NETWORK
TITLE = 218 - LCP81_C311_BG6314 - Compactor Lock In Pos. OS - Locked

       CALL #"LCP81_C311_BG6314"
       (
         CM_No := 218 ,
         Tab := 26 ,
         SubTab := 7 ,
         CfgType := 0 ,
         CfgInvert := True ,
         InputRaw := LCP81_C311_BG6314_DI_FbP ,
         SC_Local := SL_26_P ,
         CM_ALM := #ALM[209] ,
       );

NETWORK
TITLE = 219 - LCP81_C311_BG6315 - Compactor Lock Out Pos. OS - Unlocked

       CALL #"LCP81_C311_BG6315"
       (
         CM_No := 219 ,
         Tab := 26 ,
         SubTab := 7 ,
         CfgType := 0 ,
         CfgInvert := True ,
         InputRaw := LCP81_C311_BG6315_DI_FbN ,
         SC_Local := SL_26_P ,
         CM_ALM := #ALM[210] ,
       );

NETWORK
TITLE = 220 - LCP81_C311_BG6316 - Compactor Lock In Pos. DS - Locked

       CALL #"LCP81_C311_BG6316"
       (
         CM_No := 220 ,
         Tab := 26 ,
         SubTab := 7 ,
         CfgType := 0 ,
         CfgInvert := True ,
         InputRaw := LCP81_C311_BG6316_DI_FbP ,
         SC_Local := SL_26_P ,
         CM_ALM := #ALM[211] ,
       );

NETWORK
TITLE = 221 - LCP81_C311_BG6317 - Compactor Lock Out Pos. DS - Unlocked

       CALL #"LCP81_C311_BG6317"
       (
         CM_No := 221 ,
         Tab := 26 ,
         SubTab := 7 ,
         CfgType := 0 ,
         CfgInvert := True ,
         InputRaw := LCP81_C311_BG6317_DI_FbN ,
         SC_Local := SL_26_P ,
         CM_ALM := #ALM[212] ,
       );

NETWORK
TITLE = 222 - LCP81_ES01_SF6136 - Emergency Stop  - Dryer 1 Ratio Box CB.81-01

       CALL #"LCP81_ES01_SF6136"
       (
         CM_No := 222 ,
         Tab := 1 ,
         SubTab := 5 ,
         CfgType := 0 ,
         CfgInvert := True ,
         InputRaw := LCP81_ES01_SF6136_DI_ChA ,
         SC_Local := SL_01 ,
         CM_ALM := #ALM[213] ,
       );

NETWORK
TITLE = 223 - LCP81_ES01_SF6137 - Emergency Stop  - Former Fan area

       CALL #"LCP81_ES01_SF6137"
       (
         CM_No := 223 ,
         Tab := 1 ,
         SubTab := 5 ,
         CfgType := 0 ,
         CfgInvert := True ,
         InputRaw := LCP81_ES01_SF6137_DI_ChA ,
         SC_Local := SL_01 ,
         CM_ALM := #ALM[214] ,
       );

NETWORK
TITLE = 224 - LCP81_ES01_SF6138 - Emergency Stop  - Former Fan area

       CALL #"LCP81_ES01_SF6138"
       (
         CM_No := 224 ,
         Tab := 1 ,
         SubTab := 5 ,
         CfgType := 0 ,
         CfgInvert := True ,
         InputRaw := LCP81_ES01_SF6138_DI_ChA ,
         SC_Local := SL_01 ,
         CM_ALM := #ALM[215] ,
       );

NETWORK
TITLE = 225 - LCP81_ES01_SF6139 - Emergency Stop  - LCP81

       CALL #"LCP81_ES01_SF6139"
       (
         CM_No := 225 ,
         Tab := 1 ,
         SubTab := 5 ,
         CfgType := 0 ,
         CfgInvert := True ,
         InputRaw := LCP81_ES01_SF6139_DI_ChA ,
         SC_Local := SL_01 ,
         CM_ALM := #ALM[216] ,
       );

NETWORK
TITLE = 226 - LCP81_DC01_FC1000 - Power Feed Module 24VDC - Status

       CALL #"LCP81_DC01_FC1000"
       (
         CM_No := 226 ,
         Tab := 13 ,
         SubTab := 5 ,
         CfgType := 0 ,
         CfgInvert := True ,
         InputRaw := LCP81_DC01_FC1000_DI_Sts ,
         SC_Local := SL_13 ,
         CM_ALM := #ALM[217] ,
       );

NETWORK
TITLE = 227 - LCP81_IO_KF1000 - Point IO - EtherNet/IP Adapter

       CALL #"LCP81_IO_KF1000"
       (
         CM_No := 227 ,
         Tab := 13 ,
         SubTab := 5 ,
         CfgType := 0 ,
         CfgInvert := True ,
         InputRaw :=  ,
         SC_Local := SL_13 ,
         CM_ALM := #ALM[218] ,
       );

NETWORK
TITLE = 228 - LCP81_IO_KF2000 - Point IO 2nd - EtherNet/IP Adapter

       CALL #"LCP81_IO_KF2000"
       (
         CM_No := 228 ,
         Tab := 13 ,
         SubTab := 5 ,
         CfgType := 0 ,
         CfgInvert := True ,
         InputRaw :=  ,
         SC_Local := SL_13 ,
         CM_ALM := #ALM[219] ,
       );

NETWORK
TITLE = 229 - LCP81_IO_KF3047 - 24V DC 8-Point Safety Input Module - SDI

       CALL #"LCP81_IO_KF3047"
       (
         CM_No := 229 ,
         Tab := 13 ,
         SubTab := 5 ,
         CfgType := 0 ,
         CfgInvert := True ,
         InputRaw :=  ,
         SC_Local := SL_13 ,
         CM_ALM := #ALM[220] ,
       );

NETWORK
TITLE = 230 - LCP81_IO_KF3048 - 24V DC 8-Point Safety Input Module - SDI

       CALL #"LCP81_IO_KF3048"
       (
         CM_No := 230 ,
         Tab := 13 ,
         SubTab := 5 ,
         CfgType := 0 ,
         CfgInvert := True ,
         InputRaw :=  ,
         SC_Local := SL_13 ,
         CM_ALM := #ALM[221] ,
       );

NETWORK
TITLE = 231 - LCP91_A110_SF6141 - Filter 1 Zone 1 - Ex doors & Estop

       CALL #"LCP91_A110_SF6141"
       (
         CM_No := 231 ,
         Tab := 1 ,
         SubTab := 3 ,
         CfgType := 0 ,
         CfgInvert := True ,
         InputRaw := LCP91_A110_SF6141_DI_ChA ,
         SC_Local := SL_01 ,
         CM_ALM := #ALM[222] ,
       );

NETWORK
TITLE = 232 - LCP91_A110_BG7712 - Filter 1 Zone 2 - Top Door

       CALL #"LCP91_A110_BG7712"
       (
         CM_No := 232 ,
         Tab := 1 ,
         SubTab := 3 ,
         CfgType := 0 ,
         CfgInvert := True ,
         InputRaw := LCP91_A110_BG7712_DI_ChA ,
         SC_Local := SL_01 ,
         CM_ALM := #ALM[223] ,
       );

NETWORK
TITLE = 233 - LCP91_A110_BG7711 - Filter 1 Zone 3 - Bottom Doors

       CALL #"LCP91_A110_BG7711"
       (
         CM_No := 233 ,
         Tab := 1 ,
         SubTab := 3 ,
         CfgType := 0 ,
         CfgInvert := True ,
         InputRaw := LCP91_A110_BG7711_DI_ChA ,
         SC_Local := SL_01 ,
         CM_ALM := #ALM[224] ,
       );

NETWORK
TITLE = 234 - LCP91_ES01_SF6142 - Emergency Stop  - LCP91

       CALL #"LCP91_ES01_SF6142"
       (
         CM_No := 234 ,
         Tab := 1 ,
         SubTab := 3 ,
         CfgType := 0 ,
         CfgInvert := True ,
         InputRaw := LCP91_ES01_SF6142_DI_ChA ,
         SC_Local := SL_01 ,
         CM_ALM := #ALM[225] ,
       );

NETWORK
TITLE = 235 - LCP91_DC01_FC1000 - Power Feed Module 24VDC - Status

       CALL #"LCP91_DC01_FC1000"
       (
         CM_No := 235 ,
         Tab := 13 ,
         SubTab := 5 ,
         CfgType := 0 ,
         CfgInvert := True ,
         InputRaw := LCP91_DC01_FC1000_DI_Sts ,
         SC_Local := SL_13 ,
         CM_ALM := #ALM[226] ,
       );

NETWORK
TITLE = 236 - LCP91_IO_KF1000 - Point IO - EtherNet/IP Adapter

       CALL #"LCP91_IO_KF1000"
       (
         CM_No := 236 ,
         Tab := 13 ,
         SubTab := 5 ,
         CfgType := 0 ,
         CfgInvert := True ,
         InputRaw :=  ,
         SC_Local := SL_13 ,
         CM_ALM := #ALM[227] ,
       );

NETWORK
TITLE = 237 - LCP91_IO_KF3015 - 24V DC 8-Point Safety Input Module - SDI

       CALL #"LCP91_IO_KF3015"
       (
         CM_No := 237 ,
         Tab := 13 ,
         SubTab := 5 ,
         CfgType := 0 ,
         CfgInvert := True ,
         InputRaw :=  ,
         SC_Local := SL_13 ,
         CM_ALM := #ALM[228] ,
       );

NETWORK
TITLE = 238 - LCP91_IO_KF3016 - 24V DC 8-Point Safety Input Module - SDI

       CALL #"LCP91_IO_KF3016"
       (
         CM_No := 238 ,
         Tab := 13 ,
         SubTab := 5 ,
         CfgType := 0 ,
         CfgInvert := True ,
         InputRaw :=  ,
         SC_Local := SL_13 ,
         CM_ALM := #ALM[229] ,
       );

NETWORK
TITLE = 239 - LCP91_IO_KF3017 - 24V DC IO Link Master Module - IO Link

       CALL #"LCP91_IO_KF3017"
       (
         CM_No := 239 ,
         Tab := 13 ,
         SubTab := 5 ,
         CfgType := 0 ,
         CfgInvert := True ,
         InputRaw :=  ,
         SC_Local := SL_13 ,
         CM_ALM := #ALM[230] ,
       );

NETWORK
TITLE = 240 - LCP92_A210_CB.A210-14 - Control Box - Baghouse Filter 2

       CALL #"LCP92_A210_CB.A210-14"
       (
         CM_No := 240 ,
         Tab := 21 ,
         SubTab := 2 ,
         CfgType := 0 ,
         CfgInvert := True ,
         InputRaw :=  ,
         SC_Local := SL_01 ,
         CM_ALM := #ALM[231] ,
       );

NETWORK
TITLE = 241 - LCP92_A210_SF6144 - Filter 2 Zone 1 - Ex doors & Estop

       CALL #"LCP92_A210_SF6144"
       (
         CM_No := 241 ,
         Tab := 1 ,
         SubTab := 3 ,
         CfgType := 0 ,
         CfgInvert := True ,
         InputRaw := LCP92_A210_SF6144_DI_ChA ,
         SC_Local := SL_01 ,
         CM_ALM := #ALM[232] ,
       );

NETWORK
TITLE = 242 - LCP92_A210_CB.A210-15 - Control Box - Baghouse Filter 2

       CALL #"LCP92_A210_CB.A210-15"
       (
         CM_No := 242 ,
         Tab := 21 ,
         SubTab := 2 ,
         CfgType := 0 ,
         CfgInvert := True ,
         InputRaw :=  ,
         SC_Local := SL_01 ,
         CM_ALM := #ALM[233] ,
       );

NETWORK
TITLE = 243 - LCP92_A210_BG7732 - Filter 2 Zone 2 - Top Door

       CALL #"LCP92_A210_BG7732"
       (
         CM_No := 243 ,
         Tab := 1 ,
         SubTab := 3 ,
         CfgType := 0 ,
         CfgInvert := True ,
         InputRaw := LCP92_A210_BG7732_DI_ChA ,
         SC_Local := SL_01 ,
         CM_ALM := #ALM[234] ,
       );

NETWORK
TITLE = 244 - LCP92_A210_BG7731 - Filter 2 Zone 3 - Bottom Doors

       CALL #"LCP92_A210_BG7731"
       (
         CM_No := 244 ,
         Tab := 1 ,
         SubTab := 3 ,
         CfgType := 0 ,
         CfgInvert := True ,
         InputRaw := LCP92_A210_BG7731_DI_ChA ,
         SC_Local := SL_01 ,
         CM_ALM := #ALM[235] ,
       );

NETWORK
TITLE = 245 - LCP92_ES01_SF6145 - Emergency Stop  - LCP92

       CALL #"LCP92_ES01_SF6145"
       (
         CM_No := 245 ,
         Tab := 1 ,
         SubTab := 3 ,
         CfgType := 0 ,
         CfgInvert := True ,
         InputRaw := LCP92_ES01_SF6145_DI_ChA ,
         SC_Local := SL_01 ,
         CM_ALM := #ALM[236] ,
       );

NETWORK
TITLE = 246 - LCP92_DC01_FC1000 - Power Feed Module 24VDC - Status

       CALL #"LCP92_DC01_FC1000"
       (
         CM_No := 246 ,
         Tab := 13 ,
         SubTab := 5 ,
         CfgType := 0 ,
         CfgInvert := True ,
         InputRaw := LCP92_DC01_FC1000_DI_Flt ,
         SC_Local := SL_13 ,
         CM_ALM := #ALM[237] ,
       );

NETWORK
TITLE = 247 - LCP92_IO_KF1000 - Point IO - EtherNet/IP Adapter

       CALL #"LCP92_IO_KF1000"
       (
         CM_No := 247 ,
         Tab := 13 ,
         SubTab := 5 ,
         CfgType := 0 ,
         CfgInvert := True ,
         InputRaw :=  ,
         SC_Local := SL_13 ,
         CM_ALM := #ALM[238] ,
       );

NETWORK
TITLE = 248 - LCP92_IO_KF3013 - 24V DC 8-Point Safety Input Module - SDI

       CALL #"LCP92_IO_KF3013"
       (
         CM_No := 248 ,
         Tab := 13 ,
         SubTab := 5 ,
         CfgType := 0 ,
         CfgInvert := True ,
         InputRaw :=  ,
         SC_Local := SL_13 ,
         CM_ALM := #ALM[239] ,
       );

NETWORK
TITLE = 249 - LCP92_IO_KF3014 - 24V DC 8-Point Safety Input Module - SDI

       CALL #"LCP92_IO_KF3014"
       (
         CM_No := 249 ,
         Tab := 13 ,
         SubTab := 5 ,
         CfgType := 0 ,
         CfgInvert := True ,
         InputRaw :=  ,
         SC_Local := SL_13 ,
         CM_ALM := #ALM[240] ,
       );

NETWORK
TITLE = 250 - LCP92_IO_KF3015 - 24V DC IO Link Master Module - IO Link

       CALL #"LCP92_IO_KF3015"
       (
         CM_No := 250 ,
         Tab := 13 ,
         SubTab := 5 ,
         CfgType := 0 ,
         CfgInvert := True ,
         InputRaw :=  ,
         SC_Local := SL_13 ,
         CM_ALM := #ALM[241] ,
       );

NETWORK
TITLE = 251 - LCP93_A171_FN3771 - Humidifier 1 Fan 1  - Motor Disconnect

       CALL #"LCP93_A171_FN3771"
       (
         CM_No := 251 ,
         Tab := 22 ,
         SubTab := 4 ,
         CfgType := 0 ,
         CfgInvert := True ,
         InputRaw := LCP93_A171_FN3771_DI_Flt ,
         SC_Local := SL_22_P ,
         CM_ALM := #ALM[242] ,
       );

NETWORK
TITLE = 252 - LCP93_A172_FN3772 - Humidifier 1 Fan 2  - Motor Disconnect

       CALL #"LCP93_A172_FN3772"
       (
         CM_No := 252 ,
         Tab := 22 ,
         SubTab := 4 ,
         CfgType := 0 ,
         CfgInvert := True ,
         InputRaw := LCP93_A172_FN3772_DI_Flt ,
         SC_Local := SL_22_P ,
         CM_ALM := #ALM[243] ,
       );

NETWORK
TITLE = 253 - LCP93_A173_FN3773 - Humidifier 1 Fan 3  - Motor Disconnect

       CALL #"LCP93_A173_FN3773"
       (
         CM_No := 253 ,
         Tab := 22 ,
         SubTab := 4 ,
         CfgType := 0 ,
         CfgInvert := True ,
         InputRaw := LCP93_A173_FN3773_DI_Flt ,
         SC_Local := SL_22_P ,
         CM_ALM := #ALM[244] ,
       );

NETWORK
TITLE = 254 - LCP93_A174_FN3774 - Humidifier 1 Fan 4  - Motor Disconnect

       CALL #"LCP93_A174_FN3774"
       (
         CM_No := 254 ,
         Tab := 22 ,
         SubTab := 4 ,
         CfgType := 0 ,
         CfgInvert := True ,
         InputRaw := LCP93_A174_FN3774_DI_Flt ,
         SC_Local := SL_22_P ,
         CM_ALM := #ALM[245] ,
       );

NETWORK
TITLE = 255 - LCP93_A191_FN3781 - Humidifier 3 Fan 1  - Motor Disconnect

       CALL #"LCP93_A191_FN3781"
       (
         CM_No := 255 ,
         Tab := 22 ,
         SubTab := 5 ,
         CfgType := 0 ,
         CfgInvert := True ,
         InputRaw := LCP93_A191_FN3781_DI_Flt ,
         SC_Local := SL_22_P ,
         CM_ALM := #ALM[246] ,
       );

NETWORK
TITLE = 256 - LCP93_A192_FN3782 - Humidifier 3 Fan 2  - Motor Disconnect

       CALL #"LCP93_A192_FN3782"
       (
         CM_No := 256 ,
         Tab := 22 ,
         SubTab := 5 ,
         CfgType := 0 ,
         CfgInvert := True ,
         InputRaw := LCP93_A192_FN3782_DI_Flt ,
         SC_Local := SL_22_P ,
         CM_ALM := #ALM[247] ,
       );

NETWORK
TITLE = 257 - LCP93_A193_FN3783 - Humidifier 3 Fan 3 - Motor Disconnect

       CALL #"LCP93_A193_FN3783"
       (
         CM_No := 257 ,
         Tab := 22 ,
         SubTab := 5 ,
         CfgType := 0 ,
         CfgInvert := True ,
         InputRaw := LCP93_A193_FN3783_DI_Flt ,
         SC_Local := SL_22_P ,
         CM_ALM := #ALM[248] ,
       );

NETWORK
TITLE = 258 - LCP93_A194_FN3784 - Humidifier 3 Fan 4 - Motor Disconnect

       CALL #"LCP93_A194_FN3784"
       (
         CM_No := 258 ,
         Tab := 22 ,
         SubTab := 5 ,
         CfgType := 0 ,
         CfgInvert := True ,
         InputRaw := LCP93_A194_FN3784_DI_Flt ,
         SC_Local := SL_22_P ,
         CM_ALM := #ALM[249] ,
       );

NETWORK
TITLE = 259 - LCP93_A271_FN3786 - Humidifier 4 Fan 1  - Motor Disconnect

       CALL #"LCP93_A271_FN3786"
       (
         CM_No := 259 ,
         Tab := 22 ,
         SubTab := 5 ,
         CfgType := 0 ,
         CfgInvert := True ,
         InputRaw := LCP93_A271_FN3786_DI_Flt ,
         SC_Local := SL_22_P ,
         CM_ALM := #ALM[250] ,
       );

NETWORK
TITLE = 260 - LCP93_A272_FN3787 - Humidifier 4 Fan 2  - Motor Disconnect

       CALL #"LCP93_A272_FN3787"
       (
         CM_No := 260 ,
         Tab := 22 ,
         SubTab := 5 ,
         CfgType := 0 ,
         CfgInvert := True ,
         InputRaw := LCP93_A272_FN3787_DI_Flt ,
         SC_Local := SL_22_P ,
         CM_ALM := #ALM[251] ,
       );

NETWORK
TITLE = 261 - LCP93_A273_FN3788 - Humidifier 4 Fan 3  - Motor Disconnect

       CALL #"LCP93_A273_FN3788"
       (
         CM_No := 261 ,
         Tab := 22 ,
         SubTab := 5 ,
         CfgType := 0 ,
         CfgInvert := True ,
         InputRaw := LCP93_A273_FN3788_DI_Flt ,
         SC_Local := SL_22_P ,
         CM_ALM := #ALM[252] ,
       );

NETWORK
TITLE = 262 - LCP93_A274_FN3789 - Humidifier 4 Fan 4 - Motor Disconnect

       CALL #"LCP93_A274_FN3789"
       (
         CM_No := 262 ,
         Tab := 22 ,
         SubTab := 5 ,
         CfgType := 0 ,
         CfgInvert := True ,
         InputRaw := LCP93_A274_FN3789_DI_Flt ,
         SC_Local := SL_22_P ,
         CM_ALM := #ALM[253] ,
       );

NETWORK
TITLE = 263 - LCP93_A281_FN3791 - Humidifier 5 Fan 1  - Motor Disconnect

       CALL #"LCP93_A281_FN3791"
       (
         CM_No := 263 ,
         Tab := 22 ,
         SubTab := 6 ,
         CfgType := 0 ,
         CfgInvert := True ,
         InputRaw := LCP93_A281_FN3791_DI_Flt ,
         SC_Local := SL_22_P ,
         CM_ALM := #ALM[254] ,
       );

NETWORK
TITLE = 264 - LCP93_A282_FN3792 - Humidifier 5 Fan 2  - Motor Disconnect

       CALL #"LCP93_A282_FN3792"
       (
         CM_No := 264 ,
         Tab := 22 ,
         SubTab := 6 ,
         CfgType := 0 ,
         CfgInvert := True ,
         InputRaw := LCP93_A282_FN3792_DI_Flt ,
         SC_Local := SL_22_P ,
         CM_ALM := #ALM[255] ,
       );

NETWORK
TITLE = 265 - LCP93_A283_FN3793 - Humidifier 5 Fan 3  - Motor Disconnect

       CALL #"LCP93_A283_FN3793"
       (
         CM_No := 265 ,
         Tab := 22 ,
         SubTab := 6 ,
         CfgType := 0 ,
         CfgInvert := True ,
         InputRaw := LCP93_A283_FN3793_DI_Flt ,
         SC_Local := SL_22_P ,
         CM_ALM := #ALM[256] ,
       );

NETWORK
TITLE = 266 - LCP93_A284_FN3794 - Humidifier 5 Fan 4  - Motor Disconnect

       CALL #"LCP93_A284_FN3794"
       (
         CM_No := 266 ,
         Tab := 22 ,
         SubTab := 6 ,
         CfgType := 0 ,
         CfgInvert := True ,
         InputRaw := LCP93_A284_FN3794_DI_Flt ,
         SC_Local := SL_22_P ,
         CM_ALM := #ALM[257] ,
       );

NETWORK
TITLE = 267 - LCP93_A291_FN3796 - Humidifier 6 Fan 1  - Motor Disconnect

       CALL #"LCP93_A291_FN3796"
       (
         CM_No := 267 ,
         Tab := 22 ,
         SubTab := 6 ,
         CfgType := 0 ,
         CfgInvert := True ,
         InputRaw := LCP93_A291_FN3796_DI_Flt ,
         SC_Local := SL_22_P ,
         CM_ALM := #ALM[258] ,
       );

NETWORK
TITLE = 268 - LCP93_A292_FN3797 - Humidifier 6 Fan 2  - Motor Disconnect

       CALL #"LCP93_A292_FN3797"
       (
         CM_No := 268 ,
         Tab := 22 ,
         SubTab := 6 ,
         CfgType := 0 ,
         CfgInvert := True ,
         InputRaw := LCP93_A292_FN3797_DI_Flt ,
         SC_Local := SL_22_P ,
         CM_ALM := #ALM[259] ,
       );

NETWORK
TITLE = 269 - LCP93_A293_FN3798 - Humidifier 6 Fan 3  - Motor Disconnect

       CALL #"LCP93_A293_FN3798"
       (
         CM_No := 269 ,
         Tab := 22 ,
         SubTab := 6 ,
         CfgType := 0 ,
         CfgInvert := True ,
         InputRaw := LCP93_A293_FN3798_DI_Flt ,
         SC_Local := SL_22_P ,
         CM_ALM := #ALM[260] ,
       );

NETWORK
TITLE = 270 - LCP93_A294_FN3799 - Humidifier 6 Fan 4 - Motor Disconnect

       CALL #"LCP93_A294_FN3799"
       (
         CM_No := 270 ,
         Tab := 22 ,
         SubTab := 6 ,
         CfgType := 0 ,
         CfgInvert := True ,
         InputRaw := LCP93_A294_FN3799_DI_Flt ,
         SC_Local := SL_22_P ,
         CM_ALM := #ALM[261] ,
       );

NETWORK
TITLE = 271 - LCP93_A170_BG7830 - Door 1 Humidifier 1 - Fan Room

       CALL #"LCP93_A170_BG7830"
       (
         CM_No := 271 ,
         Tab := 1 ,
         SubTab := 3 ,
         CfgType := 0 ,
         CfgInvert := True ,
         InputRaw := LCP93_A170_BG7830_DI_ChA ,
         SC_Local := SL_22_P ,
         CM_ALM := #ALM[262] ,
       );

NETWORK
TITLE = 272 - LCP93_A190_BG7832 - Door 1 Humidifier 3 - Fan Room

       CALL #"LCP93_A190_BG7832"
       (
         CM_No := 272 ,
         Tab := 1 ,
         SubTab := 3 ,
         CfgType := 0 ,
         CfgInvert := True ,
         InputRaw := LCP93_A190_BG7832_DI_ChA ,
         SC_Local := SL_22_P ,
         CM_ALM := #ALM[263] ,
       );

NETWORK
TITLE = 273 - LCP93_A270_BG7834 - Door 1 Humidifier 4 - Fan Room

       CALL #"LCP93_A270_BG7834"
       (
         CM_No := 273 ,
         Tab := 1 ,
         SubTab := 3 ,
         CfgType := 0 ,
         CfgInvert := True ,
         InputRaw := LCP93_A270_BG7834_DI_ChA ,
         SC_Local := SL_22_P ,
         CM_ALM := #ALM[264] ,
       );

NETWORK
TITLE = 274 - LCP93_A280_BG7836 - Door 1 Humidifier 5 - Fan Room

       CALL #"LCP93_A280_BG7836"
       (
         CM_No := 274 ,
         Tab := 1 ,
         SubTab := 3 ,
         CfgType := 0 ,
         CfgInvert := True ,
         InputRaw := LCP93_A280_BG7836_DI_ChA ,
         SC_Local := SL_22_P ,
         CM_ALM := #ALM[265] ,
       );

NETWORK
TITLE = 275 - LCP93_A290_BG7838 - Door 1 Humidifier 6 - Fan Room

       CALL #"LCP93_A290_BG7838"
       (
         CM_No := 275 ,
         Tab := 1 ,
         SubTab := 3 ,
         CfgType := 0 ,
         CfgInvert := True ,
         InputRaw := LCP93_A290_BG7838_DI_ChA ,
         SC_Local := SL_22_P ,
         CM_ALM := #ALM[266] ,
       );

NETWORK
TITLE = 276 - LCP93_ES01_SF6146 - Emergency Stop  - Humidifier Area

       CALL #"LCP93_ES01_SF6146"
       (
         CM_No := 276 ,
         Tab := 1 ,
         SubTab := 3 ,
         CfgType := 0 ,
         CfgInvert := True ,
         InputRaw := LCP93_ES01_SF6146_DI_ChA ,
         SC_Local := SL_01 ,
         CM_ALM := #ALM[267] ,
       );

NETWORK
TITLE = 277 - LCP93_ES01_SF6147 - Emergency Stop  - Humidifier Area

       CALL #"LCP93_ES01_SF6147"
       (
         CM_No := 277 ,
         Tab := 1 ,
         SubTab := 3 ,
         CfgType := 0 ,
         CfgInvert := True ,
         InputRaw := LCP93_ES01_SF6147_DI_ChA ,
         SC_Local := SL_01 ,
         CM_ALM := #ALM[268] ,
       );

NETWORK
TITLE = 278 - LCP93_ES01_SF6148 - Emergency Stop  - Humidifier Area

       CALL #"LCP93_ES01_SF6148"
       (
         CM_No := 278 ,
         Tab := 1 ,
         SubTab := 3 ,
         CfgType := 0 ,
         CfgInvert := True ,
         InputRaw := LCP93_ES01_SF6148_DI_ChA ,
         SC_Local := SL_01 ,
         CM_ALM := #ALM[269] ,
       );

NETWORK
TITLE = 279 - LCP93_ES01_SF6149 - Emergency Stop  - LCP93

       CALL #"LCP93_ES01_SF6149"
       (
         CM_No := 279 ,
         Tab := 1 ,
         SubTab := 3 ,
         CfgType := 0 ,
         CfgInvert := True ,
         InputRaw := LCP93_ES01_SF6149_DI_ChA ,
         SC_Local := SL_01 ,
         CM_ALM := #ALM[270] ,
       );

NETWORK
TITLE = 280 - LCP93_DC01_FC1000 - Power Feed Module 24VDC - Status

       CALL #"LCP93_DC01_FC1000"
       (
         CM_No := 280 ,
         Tab := 13 ,
         SubTab := 5 ,
         CfgType := 0 ,
         CfgInvert := True ,
         InputRaw := LCP93_DC01_FC1000_DI_Flt ,
         SC_Local := SL_13 ,
         CM_ALM := #ALM[271] ,
       );

NETWORK
TITLE = 281 - LCP93_IO_KF1000 - Point IO - EtherNet/IP Adapter

       CALL #"LCP93_IO_KF1000"
       (
         CM_No := 281 ,
         Tab := 13 ,
         SubTab := 5 ,
         CfgType := 0 ,
         CfgInvert := True ,
         InputRaw :=  ,
         SC_Local := SL_13 ,
         CM_ALM := #ALM[272] ,
       );

NETWORK
TITLE = 282 - LCP93_IO_KF3020 - 24V DC 8-Point Safety Input Module - SDI

       CALL #"LCP93_IO_KF3020"
       (
         CM_No := 282 ,
         Tab := 13 ,
         SubTab := 5 ,
         CfgType := 0 ,
         CfgInvert := True ,
         InputRaw :=  ,
         SC_Local := SL_13 ,
         CM_ALM := #ALM[273] ,
       );

NETWORK
TITLE = 283 - LCP93_IO_KF3021 - 24V DC 8-Point Safety Input Module - SDI

       CALL #"LCP93_IO_KF3021"
       (
         CM_No := 283 ,
         Tab := 13 ,
         SubTab := 5 ,
         CfgType := 0 ,
         CfgInvert := True ,
         InputRaw :=  ,
         SC_Local := SL_13 ,
         CM_ALM := #ALM[274] ,
       );

NETWORK
TITLE = 284 - LCP93_IO_KF3022 - 24V DC 8-Point Safety Input Module - SDI

       CALL #"LCP93_IO_KF3022"
       (
         CM_No := 284 ,
         Tab := 13 ,
         SubTab := 5 ,
         CfgType := 0 ,
         CfgInvert := True ,
         InputRaw :=  ,
         SC_Local := SL_13 ,
         CM_ALM := #ALM[275] ,
       );

NETWORK
TITLE = 285 - LCP101_AC01_FC3101 - 115VAC Power Supply - Thermal Fault

       CALL #"LCP101_AC01_FC3101"
       (
         CM_No := 285 ,
         Tab := 13 ,
         SubTab := 6 ,
         CfgType := 0 ,
         CfgInvert := True ,
         InputRaw := LCP101_AC01_FC3101_DI_Flt ,
         SC_Local := SL_13 ,
         CM_ALM := #ALM[276] ,
       );

NETWORK
TITLE = 286 - LCP101_I610_QA1101 - Min Gas Pressure Switch - (-BP8101)

       CALL #"LCP101_I610_QA1101"
       (
         CM_No := 286 ,
         Tab := 28 ,
         SubTab := 3 ,
         CfgType := 0 ,
         CfgInvert := True ,
         InputRaw := LCP101_I610_QA1101_DI_FltL ,
         SC_Local := SL_28_S1 ,
         CM_ALM := #ALM[277] ,
       );

NETWORK
TITLE = 287 - LCP101_I610_QA1102 - Max Gas Pressure Switch - (-BP8102)

       CALL #"LCP101_I610_QA1102"
       (
         CM_No := 287 ,
         Tab := 28 ,
         SubTab := 3 ,
         CfgType := 0 ,
         CfgInvert := True ,
         InputRaw := LCP101_I610_QA1102_DI_FltH ,
         SC_Local := SL_28_S1 ,
         CM_ALM := #ALM[278] ,
       );

NETWORK
TITLE = 288 - LCP101_I610_QA1103 - Leak Gas Pressure Switch - (-BP8103)

       CALL #"LCP101_I610_QA1103"
       (
         CM_No := 288 ,
         Tab := 28 ,
         SubTab := 3 ,
         CfgType := 0 ,
         CfgInvert := True ,
         InputRaw := LCP101_I610_QA1103_DI_Ps ,
         SC_Local := SL_28_S1 ,
         CM_ALM := #ALM[279] ,
       );

NETWORK
TITLE = 289 - LCP101_I610_QA1113 - No Air Check Pressure Switch - (-BP2113)

       CALL #"LCP101_I610_QA1113"
       (
         CM_No := 289 ,
         Tab := 28 ,
         SubTab := 3 ,
         CfgType := 0 ,
         CfgInvert := True ,
         InputRaw := LCP101_I610_QA1113_DI_Ps ,
         SC_Local := SL_28_S1 ,
         CM_ALM := #ALM[280] ,
       );

NETWORK
TITLE = 290 - LCP101_I610_QA1108 - Burner Failure - Signal from Maxon

       CALL #"LCP101_I610_QA1108"
       (
         CM_No := 290 ,
         Tab := 28 ,
         SubTab := 3 ,
         CfgType := 0 ,
         CfgInvert := True ,
         InputRaw := LCP101_I610_QA1108_DI_Flt ,
         SC_Local := SL_28_S1 ,
         CM_ALM := #ALM[281] ,
       );

NETWORK
TITLE = 291 - LCP101_I610_QA1104 - High Temperature Failure - Signal from JUMO

       CALL #"LCP101_I610_QA1104"
       (
         CM_No := 291 ,
         Tab := 28 ,
         SubTab := 3 ,
         CfgType := 0 ,
         CfgInvert := True ,
         InputRaw := LCP101_I610_QA1104_DI_Flt ,
         SC_Local := SL_28_S1 ,
         CM_ALM := #ALM[282] ,
       );

NETWORK
TITLE = 292 - LCP101_I512_BG7101 - Disc Filter 1 Door 1 - Before Filter

       CALL #"LCP101_I512_BG7101"
       (
         CM_No := 292 ,
         Tab := 1 ,
         SubTab := 8 ,
         CfgType := 0 ,
         CfgInvert := True ,
         InputRaw := LCP101_I512_BG7101_DI_ChA ,
         SC_Local := SL_28_S1 ,
         CM_ALM := #ALM[283] ,
       );

NETWORK
TITLE = 293 - LCP101_I512_BG7103 - Disc Filter 1 Door 2 - After Filter

       CALL #"LCP101_I512_BG7103"
       (
         CM_No := 293 ,
         Tab := 1 ,
         SubTab := 8 ,
         CfgType := 0 ,
         CfgInvert := True ,
         InputRaw := LCP101_I512_BG7103_DI_ChA ,
         SC_Local := SL_28_S1 ,
         CM_ALM := #ALM[284] ,
       );

NETWORK
TITLE = 294 - LCP101_I611_BP1120 - Zone 1 Circulation Fan - Diff. Pressure Circ. Fan 1

       CALL #"LCP101_I611_BP1120"
       (
         CM_No := 294 ,
         Tab := 28 ,
         SubTab := 3 ,
         CfgType := 0 ,
         CfgInvert := True ,
         InputRaw := LCP101_I611_BP1120_DI_Ps ,
         SC_Local := SL_28_S1 ,
         CM_ALM := #ALM[285] ,
       );

NETWORK
TITLE = 295 - LCP101_ES01_SF6151 - Emergency Stop  - Dryer 1 Zone 1 Area

       CALL #"LCP101_ES01_SF6151"
       (
         CM_No := 295 ,
         Tab := 1 ,
         SubTab := 5 ,
         CfgType := 0 ,
         CfgInvert := True ,
         InputRaw := LCP101_ES01_SF6151_DI_ChA ,
         SC_Local := SL_01 ,
         CM_ALM := #ALM[286] ,
       );

NETWORK
TITLE = 296 - LCP101_ES01_SF6152 - Emergency Stop  - LCP101

       CALL #"LCP101_ES01_SF6152"
       (
         CM_No := 296 ,
         Tab := 1 ,
         SubTab := 5 ,
         CfgType := 0 ,
         CfgInvert := True ,
         InputRaw := LCP101_ES01_SF6152_DI_ChA ,
         SC_Local := SL_01 ,
         CM_ALM := #ALM[287] ,
       );

NETWORK
TITLE = 297 - LCP101_DC01_FC1000 - Power Feed Module 24VDC - Status

       CALL #"LCP101_DC01_FC1000"
       (
         CM_No := 297 ,
         Tab := 13 ,
         SubTab := 6 ,
         CfgType := 0 ,
         CfgInvert := True ,
         InputRaw := LCP101_DC01_FC1000_DI_Flt ,
         SC_Local := SL_13 ,
         CM_ALM := #ALM[288] ,
       );

NETWORK
TITLE = 298 - LCP101_IO_KF1000 - Point IO - EtherNet/IP Adapter

       CALL #"LCP101_IO_KF1000"
       (
         CM_No := 298 ,
         Tab := 13 ,
         SubTab := 6 ,
         CfgType := 0 ,
         CfgInvert := True ,
         InputRaw :=  ,
         SC_Local := SL_13 ,
         CM_ALM := #ALM[289] ,
       );

NETWORK
TITLE = 299 - LCP101_IO_KF3013 - 24V DC 8-Point Safety Input Module - SDI

       CALL #"LCP101_IO_KF3013"
       (
         CM_No := 299 ,
         Tab := 13 ,
         SubTab := 6 ,
         CfgType := 0 ,
         CfgInvert := True ,
         InputRaw :=  ,
         SC_Local := SL_13 ,
         CM_ALM := #ALM[290] ,
       );

NETWORK
TITLE = 300 - LCP101_IO_KF3014 - 24V DC 8-Point Safety Input Module - SDI

       CALL #"LCP101_IO_KF3014"
       (
         CM_No := 300 ,
         Tab := 13 ,
         SubTab := 6 ,
         CfgType := 0 ,
         CfgInvert := True ,
         InputRaw :=  ,
         SC_Local := SL_13 ,
         CM_ALM := #ALM[291] ,
       );

NETWORK
TITLE = 301 - LCP102_AC01_FC3201 - 115VAC Power Supply - Thermal Fault

       CALL #"LCP102_AC01_FC3201"
       (
         CM_No := 301 ,
         Tab := 13 ,
         SubTab := 6 ,
         CfgType := 0 ,
         CfgInvert := True ,
         InputRaw := LCP102_AC01_FC3201_DI_Flt ,
         SC_Local := SL_13 ,
         CM_ALM := #ALM[292] ,
       );

NETWORK
TITLE = 302 - LCP102_I522_BG7201 - Disc Filter 2 Door 1 - Before Filter

       CALL #"LCP102_I522_BG7201"
       (
         CM_No := 302 ,
         Tab := 1 ,
         SubTab := 8 ,
         CfgType := 0 ,
         CfgInvert := True ,
         InputRaw := LCP102_I522_BG7201_DI_ChA ,
         SC_Local := SL_28_S1 ,
         CM_ALM := #ALM[293] ,
       );

NETWORK
TITLE = 303 - LCP102_I522_BG7203 - Disc Filter 2 Door 1 - After Filter

       CALL #"LCP102_I522_BG7203"
       (
         CM_No := 303 ,
         Tab := 1 ,
         SubTab := 8 ,
         CfgType := 0 ,
         CfgInvert := True ,
         InputRaw := LCP102_I522_BG7203_DI_ChA ,
         SC_Local := SL_28_S1 ,
         CM_ALM := #ALM[294] ,
       );

NETWORK
TITLE = 304 - LCP102_I621_BP1222 - Zone 2 Circulation Fan - Diff. Pressure Circ. Fan 2

       CALL #"LCP102_I621_BP1222"
       (
         CM_No := 304 ,
         Tab := 28 ,
         SubTab := 4 ,
         CfgType := 0 ,
         CfgInvert := True ,
         InputRaw := LCP102_I621_BP1222_DI_Ps ,
         SC_Local := SL_28_S1 ,
         CM_ALM := #ALM[295] ,
       );

NETWORK
TITLE = 305 - LCP102_ES01_SF6253 - Emergency Stop  - Dryer 1 Zone 2 Area

       CALL #"LCP102_ES01_SF6253"
       (
         CM_No := 305 ,
         Tab := 1 ,
         SubTab := 5 ,
         CfgType := 0 ,
         CfgInvert := True ,
         InputRaw := LCP102_ES01_SF6253_DI_ChA ,
         SC_Local := SL_01 ,
         CM_ALM := #ALM[296] ,
       );

NETWORK
TITLE = 306 - LCP102_ES01_SF6254 - Emergency Stop  - LCP102

       CALL #"LCP102_ES01_SF6254"
       (
         CM_No := 306 ,
         Tab := 1 ,
         SubTab := 5 ,
         CfgType := 0 ,
         CfgInvert := True ,
         InputRaw := LCP102_ES01_SF6254_DI_ChA ,
         SC_Local := SL_01 ,
         CM_ALM := #ALM[297] ,
       );

NETWORK
TITLE = 307 - LCP102_DC01_FC1000 - Power Feed Module 24VDC - Status

       CALL #"LCP102_DC01_FC1000"
       (
         CM_No := 307 ,
         Tab := 13 ,
         SubTab := 6 ,
         CfgType := 0 ,
         CfgInvert := True ,
         InputRaw := LCP102_DC01_FC1000_DI_Flt ,
         SC_Local := SL_13 ,
         CM_ALM := #ALM[298] ,
       );

NETWORK
TITLE = 308 - LCP102_IO_KF1000 - Point IO - EtherNet/IP Adapter

       CALL #"LCP102_IO_KF1000"
       (
         CM_No := 308 ,
         Tab := 13 ,
         SubTab := 6 ,
         CfgType := 0 ,
         CfgInvert := True ,
         InputRaw :=  ,
         SC_Local := SL_13 ,
         CM_ALM := #ALM[299] ,
       );

NETWORK
TITLE = 309 - LCP102_IO_KF3008 - 24V DC 8-Point Safety Input Module - SDI

       CALL #"LCP102_IO_KF3008"
       (
         CM_No := 309 ,
         Tab := 13 ,
         SubTab := 6 ,
         CfgType := 0 ,
         CfgInvert := True ,
         InputRaw :=  ,
         SC_Local := SL_13 ,
         CM_ALM := #ALM[300] ,
       );

NETWORK
TITLE = 310 - LCP102_IO_KF3009 - 24V DC 8-Point Safety Input Module - SDI

       CALL #"LCP102_IO_KF3009"
       (
         CM_No := 310 ,
         Tab := 13 ,
         SubTab := 6 ,
         CfgType := 0 ,
         CfgInvert := True ,
         InputRaw :=  ,
         SC_Local := SL_13 ,
         CM_ALM := #ALM[301] ,
       );

NETWORK
TITLE = 311 - LCP102_IO_KF3010 - 24V DC 8-Point Source Safety Output Module - SDO

       CALL #"LCP102_IO_KF3010"
       (
         CM_No := 311 ,
         Tab := 13 ,
         SubTab := 6 ,
         CfgType := 0 ,
         CfgInvert := True ,
         InputRaw :=  ,
         SC_Local := SL_13 ,
         CM_ALM := #ALM[302] ,
       );

NETWORK
TITLE = 312 - LCP103_AC01_FC3301 - 115VAC Power Supply - Thermal Fault

       CALL #"LCP103_AC01_FC3301"
       (
         CM_No := 312 ,
         Tab := 13 ,
         SubTab := 6 ,
         CfgType := 0 ,
         CfgInvert := True ,
         InputRaw := LCP103_AC01_FC3301_DI_Flt ,
         SC_Local := SL_13 ,
         CM_ALM := #ALM[303] ,
       );

NETWORK
TITLE = 313 - LCP103_I630_QA1301 - Min Gas Pressure Switch - (-BP8301)

       CALL #"LCP103_I630_QA1301"
       (
         CM_No := 313 ,
         Tab := 28 ,
         SubTab := 5 ,
         CfgType := 0 ,
         CfgInvert := True ,
         InputRaw := LCP103_I630_QA1301_DI_FltL ,
         SC_Local := SL_28_S2 ,
         CM_ALM := #ALM[304] ,
       );

NETWORK
TITLE = 314 - LCP103_I630_QA1302 - Max Gas Pressure Switch - (-BP8302)

       CALL #"LCP103_I630_QA1302"
       (
         CM_No := 314 ,
         Tab := 28 ,
         SubTab := 5 ,
         CfgType := 0 ,
         CfgInvert := True ,
         InputRaw := LCP103_I630_QA1302_DI_FltH ,
         SC_Local := SL_28_S2 ,
         CM_ALM := #ALM[305] ,
       );

NETWORK
TITLE = 315 - LCP103_I630_QA1303 - Leak Gas Pressure Switch - (-BP8303)

       CALL #"LCP103_I630_QA1303"
       (
         CM_No := 315 ,
         Tab := 28 ,
         SubTab := 5 ,
         CfgType := 0 ,
         CfgInvert := True ,
         InputRaw := LCP103_I630_QA1303_DI_Ps ,
         SC_Local := SL_28_S2 ,
         CM_ALM := #ALM[306] ,
       );

NETWORK
TITLE = 316 - LCP103_I630_QA1313 - No Air Check Pressure Switch - (-BP2313)

       CALL #"LCP103_I630_QA1313"
       (
         CM_No := 316 ,
         Tab := 28 ,
         SubTab := 5 ,
         CfgType := 0 ,
         CfgInvert := True ,
         InputRaw := LCP103_I630_QA1313_DI_Ps ,
         SC_Local := SL_28_S2 ,
         CM_ALM := #ALM[307] ,
       );

NETWORK
TITLE = 317 - LCP103_I630_QA1308 - Burner Failure - Signal from Maxon

       CALL #"LCP103_I630_QA1308"
       (
         CM_No := 317 ,
         Tab := 28 ,
         SubTab := 5 ,
         CfgType := 0 ,
         CfgInvert := True ,
         InputRaw := LCP103_I630_QA1308_DI_Flt ,
         SC_Local := SL_28_S2 ,
         CM_ALM := #ALM[308] ,
       );

NETWORK
TITLE = 318 - LCP103_I630_QA1304 - High Temperature Failure - Signal from JUMO

       CALL #"LCP103_I630_QA1304"
       (
         CM_No := 318 ,
         Tab := 28 ,
         SubTab := 5 ,
         CfgType := 0 ,
         CfgInvert := True ,
         InputRaw := LCP103_I630_QA1304_DI_Flt ,
         SC_Local := SL_28_S2 ,
         CM_ALM := #ALM[309] ,
       );

NETWORK
TITLE = 319 - LCP103_K512_BG7301 - Disc Filter 3 Door 1 - Before Filter

       CALL #"LCP103_K512_BG7301"
       (
         CM_No := 319 ,
         Tab := 1 ,
         SubTab := 8 ,
         CfgType := 0 ,
         CfgInvert := True ,
         InputRaw := LCP103_K512_BG7301_DI_ChA ,
         SC_Local := SL_28_S2 ,
         CM_ALM := #ALM[310] ,
       );

NETWORK
TITLE = 320 - LCP103_K512_BG7303 - Disc Filter 3 Door 2 - After Filter

       CALL #"LCP103_K512_BG7303"
       (
         CM_No := 320 ,
         Tab := 1 ,
         SubTab := 8 ,
         CfgType := 0 ,
         CfgInvert := True ,
         InputRaw := LCP103_K512_BG7303_DI_ChA ,
         SC_Local := SL_28_S2 ,
         CM_ALM := #ALM[311] ,
       );

NETWORK
TITLE = 321 - LCP103_K611_BP1323 - Zone 3 Circulation Fan - Diff. Pressure Circ. Fan 3

       CALL #"LCP103_K611_BP1323"
       (
         CM_No := 321 ,
         Tab := 28 ,
         SubTab := 5 ,
         CfgType := 0 ,
         CfgInvert := True ,
         InputRaw := LCP103_K611_BP1323_DI_Ps ,
         SC_Local := SL_28_S2 ,
         CM_ALM := #ALM[312] ,
       );

NETWORK
TITLE = 322 - LCP103_ES01_SF6355 - Emergency Stop  - Dryer 2 Zone 3 Area

       CALL #"LCP103_ES01_SF6355"
       (
         CM_No := 322 ,
         Tab := 1 ,
         SubTab := 5 ,
         CfgType := 0 ,
         CfgInvert := True ,
         InputRaw := LCP103_ES01_SF6355_DI_ChA ,
         SC_Local := SL_01 ,
         CM_ALM := #ALM[313] ,
       );

NETWORK
TITLE = 323 - LCP103_ES01_SF6356 - Emergency Stop  - LCP103

       CALL #"LCP103_ES01_SF6356"
       (
         CM_No := 323 ,
         Tab := 1 ,
         SubTab := 5 ,
         CfgType := 0 ,
         CfgInvert := True ,
         InputRaw := LCP103_ES01_SF6356_DI_ChA ,
         SC_Local := SL_01 ,
         CM_ALM := #ALM[314] ,
       );

NETWORK
TITLE = 324 - LCP103_DC01_FC1000 - Power Feed Module 24VDC - Status

       CALL #"LCP103_DC01_FC1000"
       (
         CM_No := 324 ,
         Tab := 13 ,
         SubTab := 6 ,
         CfgType := 0 ,
         CfgInvert := True ,
         InputRaw := LCP103_DC01_FC1000_DI_Flt ,
         SC_Local := SL_13 ,
         CM_ALM := #ALM[315] ,
       );

NETWORK
TITLE = 325 - LCP103_IO_KF1000 - Point IO - EtherNet/IP Adapter

       CALL #"LCP103_IO_KF1000"
       (
         CM_No := 325 ,
         Tab := 13 ,
         SubTab := 6 ,
         CfgType := 0 ,
         CfgInvert := True ,
         InputRaw :=  ,
         SC_Local := SL_13 ,
         CM_ALM := #ALM[316] ,
       );

NETWORK
TITLE = 326 - LCP103_IO_KF3013 - 24V DC 8-Point Safety Input Module - SDI

       CALL #"LCP103_IO_KF3013"
       (
         CM_No := 326 ,
         Tab := 13 ,
         SubTab := 6 ,
         CfgType := 0 ,
         CfgInvert := True ,
         InputRaw :=  ,
         SC_Local := SL_13 ,
         CM_ALM := #ALM[317] ,
       );

NETWORK
TITLE = 327 - LCP103_IO_KF3014 - 24V DC 8-Point Safety Input Module - SDI

       CALL #"LCP103_IO_KF3014"
       (
         CM_No := 327 ,
         Tab := 13 ,
         SubTab := 6 ,
         CfgType := 0 ,
         CfgInvert := True ,
         InputRaw :=  ,
         SC_Local := SL_13 ,
         CM_ALM := #ALM[318] ,
       );

NETWORK
TITLE = 328 - LCP104_AC01_FC3401 - 115VAC Power Supply - Thermal Fault

       CALL #"LCP104_AC01_FC3401"
       (
         CM_No := 328 ,
         Tab := 13 ,
         SubTab := 6 ,
         CfgType := 0 ,
         CfgInvert := True ,
         InputRaw := LCP104_AC01_FC3401_DI_Flt ,
         SC_Local := SL_13 ,
         CM_ALM := #ALM[319] ,
       );

NETWORK
TITLE = 329 - LCP104_I640_QA1401 - Min Gas Pressure Switch - (-BP8401)

       CALL #"LCP104_I640_QA1401"
       (
         CM_No := 329 ,
         Tab := 28 ,
         SubTab := 6 ,
         CfgType := 0 ,
         CfgInvert := True ,
         InputRaw := LCP104_I640_QA1401_DI_FltL ,
         SC_Local := SL_28_S2 ,
         CM_ALM := #ALM[320] ,
       );

NETWORK
TITLE = 330 - LCP104_I640_QA1402 - Max Gas Pressure Switch - (-BP8402)

       CALL #"LCP104_I640_QA1402"
       (
         CM_No := 330 ,
         Tab := 28 ,
         SubTab := 6 ,
         CfgType := 0 ,
         CfgInvert := True ,
         InputRaw := LCP104_I640_QA1402_DI_FltH ,
         SC_Local := SL_28_S2 ,
         CM_ALM := #ALM[321] ,
       );

NETWORK
TITLE = 331 - LCP104_I640_QA1403 - Leak Gas Pressure Switch - (-BP8403)

       CALL #"LCP104_I640_QA1403"
       (
         CM_No := 331 ,
         Tab := 28 ,
         SubTab := 6 ,
         CfgType := 0 ,
         CfgInvert := True ,
         InputRaw := LCP104_I640_QA1403_DI_Ps ,
         SC_Local := SL_28_S2 ,
         CM_ALM := #ALM[322] ,
       );

NETWORK
TITLE = 332 - LCP104_I640_QA1413 - No Air Check Pressure Switch - (-BP2413)

       CALL #"LCP104_I640_QA1413"
       (
         CM_No := 332 ,
         Tab := 28 ,
         SubTab := 6 ,
         CfgType := 0 ,
         CfgInvert := True ,
         InputRaw := LCP104_I640_QA1413_DI_Ps ,
         SC_Local := SL_28_S2 ,
         CM_ALM := #ALM[323] ,
       );

NETWORK
TITLE = 333 - LCP104_I640_QA1408 - Burner Failure - Signal from Maxon

       CALL #"LCP104_I640_QA1408"
       (
         CM_No := 333 ,
         Tab := 28 ,
         SubTab := 6 ,
         CfgType := 0 ,
         CfgInvert := True ,
         InputRaw := LCP104_I640_QA1408_DI_Flt ,
         SC_Local := SL_28_S2 ,
         CM_ALM := #ALM[324] ,
       );

NETWORK
TITLE = 334 - LCP104_I640_QA1404 - High Temperature Failure - Signal from JUMO

       CALL #"LCP104_I640_QA1404"
       (
         CM_No := 334 ,
         Tab := 28 ,
         SubTab := 6 ,
         CfgType := 0 ,
         CfgInvert := True ,
         InputRaw := LCP104_I640_QA1404_DI_Flt ,
         SC_Local := SL_28_S2 ,
         CM_ALM := #ALM[325] ,
       );

NETWORK
TITLE = 335 - LCP104_K522_BG7401 - Disc Filter 4 Door 1 - Before Filter

       CALL #"LCP104_K522_BG7401"
       (
         CM_No := 335 ,
         Tab := 1 ,
         SubTab := 8 ,
         CfgType := 0 ,
         CfgInvert := True ,
         InputRaw := LCP104_K522_BG7401_DI_ChA ,
         SC_Local := SL_28_S2 ,
         CM_ALM := #ALM[326] ,
       );

NETWORK
TITLE = 336 - LCP104_K522_BG7403 - Disc Filter 4 Door 2 - After Filter

       CALL #"LCP104_K522_BG7403"
       (
         CM_No := 336 ,
         Tab := 1 ,
         SubTab := 8 ,
         CfgType := 0 ,
         CfgInvert := True ,
         InputRaw := LCP104_K522_BG7403_DI_ChA ,
         SC_Local := SL_28_S2 ,
         CM_ALM := #ALM[327] ,
       );

NETWORK
TITLE = 337 - LCP104_K621_BP1424 - Zone 4 Circulation Fan  - Diff. Pressure Circ. Fan 4

       CALL #"LCP104_K621_BP1424"
       (
         CM_No := 337 ,
         Tab := 28 ,
         SubTab := 6 ,
         CfgType := 0 ,
         CfgInvert := True ,
         InputRaw := LCP104_K621_BP1424_DI_Ps ,
         SC_Local := SL_28_S2 ,
         CM_ALM := #ALM[328] ,
       );

NETWORK
TITLE = 338 - LCP104_ES01_SF6457 - Emergency Stop  - Dryer 2 Zone 4 Area

       CALL #"LCP104_ES01_SF6457"
       (
         CM_No := 338 ,
         Tab := 1 ,
         SubTab := 5 ,
         CfgType := 0 ,
         CfgInvert := True ,
         InputRaw := LCP104_ES01_SF6457_DI_ChA ,
         SC_Local := SL_01 ,
         CM_ALM := #ALM[329] ,
       );

NETWORK
TITLE = 339 - LCP104_ES01_SF6458 - Emergency Stop  - LCP104

       CALL #"LCP104_ES01_SF6458"
       (
         CM_No := 339 ,
         Tab := 1 ,
         SubTab := 5 ,
         CfgType := 0 ,
         CfgInvert := True ,
         InputRaw := LCP104_ES01_SF6458_DI_ChA ,
         SC_Local := SL_01 ,
         CM_ALM := #ALM[330] ,
       );

NETWORK
TITLE = 340 - LCP104_DC01_FC1000 - Power Feed Module 24VDC - Status

       CALL #"LCP104_DC01_FC1000"
       (
         CM_No := 340 ,
         Tab := 13 ,
         SubTab := 6 ,
         CfgType := 0 ,
         CfgInvert := True ,
         InputRaw := LCP104_DC01_FC1000_DI_Flt ,
         SC_Local := SL_13 ,
         CM_ALM := #ALM[331] ,
       );

NETWORK
TITLE = 341 - LCP104_IO_KF1000 - Point IO - EtherNet/IP Adapter

       CALL #"LCP104_IO_KF1000"
       (
         CM_No := 341 ,
         Tab := 13 ,
         SubTab := 6 ,
         CfgType := 0 ,
         CfgInvert := True ,
         InputRaw :=  ,
         SC_Local := SL_13 ,
         CM_ALM := #ALM[332] ,
       );

NETWORK
TITLE = 342 - LCP104_IO_KF3013 - 24V DC 8-Point Safety Input Module - SDI

       CALL #"LCP104_IO_KF3013"
       (
         CM_No := 342 ,
         Tab := 13 ,
         SubTab := 6 ,
         CfgType := 0 ,
         CfgInvert := True ,
         InputRaw :=  ,
         SC_Local := SL_13 ,
         CM_ALM := #ALM[333] ,
       );

NETWORK
TITLE = 343 - LCP104_IO_KF3014 - 24V DC 8-Point Safety Input Module - SDI

       CALL #"LCP104_IO_KF3014"
       (
         CM_No := 343 ,
         Tab := 13 ,
         SubTab := 6 ,
         CfgType := 0 ,
         CfgInvert := True ,
         InputRaw :=  ,
         SC_Local := SL_13 ,
         CM_ALM := #ALM[334] ,
       );

NETWORK
TITLE = 344 - LCP111_AC01_FC3501 - 115VAC Power Supply - Thermal Fault

       CALL #"LCP111_AC01_FC3501"
       (
         CM_No := 344 ,
         Tab := 13 ,
         SubTab := 6 ,
         CfgType := 0 ,
         CfgInvert := True ,
         InputRaw := LCP111_AC01_FC3501_DI_Flt ,
         SC_Local := SL_13 ,
         CM_ALM := #ALM[335] ,
       );

NETWORK
TITLE = 345 - LCP111_I650_QA1501 - Min Gas Pressure Switch - (-BP8501)

       CALL #"LCP111_I650_QA1501"
       (
         CM_No := 345 ,
         Tab := 28 ,
         SubTab := 7 ,
         CfgType := 0 ,
         CfgInvert := True ,
         InputRaw := LCP111_I650_QA1501_DI_FltL ,
         SC_Local := SL_28_S3 ,
         CM_ALM := #ALM[336] ,
       );

NETWORK
TITLE = 346 - LCP111_I650_QA1502 - Max Gas Pressure Switch - (-BP8502)

       CALL #"LCP111_I650_QA1502"
       (
         CM_No := 346 ,
         Tab := 28 ,
         SubTab := 7 ,
         CfgType := 0 ,
         CfgInvert := True ,
         InputRaw := LCP111_I650_QA1502_DI_FltH ,
         SC_Local := SL_28_S3 ,
         CM_ALM := #ALM[337] ,
       );

NETWORK
TITLE = 347 - LCP111_I650_QA1503 - Leak Gas Pressure Switch - (-BP8503)

       CALL #"LCP111_I650_QA1503"
       (
         CM_No := 347 ,
         Tab := 28 ,
         SubTab := 7 ,
         CfgType := 0 ,
         CfgInvert := True ,
         InputRaw := LCP111_I650_QA1503_DI_Ps ,
         SC_Local := SL_28_S3 ,
         CM_ALM := #ALM[338] ,
       );

NETWORK
TITLE = 348 - LCP111_I650_QA1513 - No Air Check Pressure Switch - (-BP2513)

       CALL #"LCP111_I650_QA1513"
       (
         CM_No := 348 ,
         Tab := 28 ,
         SubTab := 7 ,
         CfgType := 0 ,
         CfgInvert := True ,
         InputRaw := LCP111_I650_QA1513_DI_Ps ,
         SC_Local := SL_28_S3 ,
         CM_ALM := #ALM[339] ,
       );

NETWORK
TITLE = 349 - LCP111_I650_QA1508 - Burner Failure - Signal from Maxon

       CALL #"LCP111_I650_QA1508"
       (
         CM_No := 349 ,
         Tab := 28 ,
         SubTab := 7 ,
         CfgType := 0 ,
         CfgInvert := True ,
         InputRaw := LCP111_I650_QA1508_DI_Flt ,
         SC_Local := SL_28_S3 ,
         CM_ALM := #ALM[340] ,
       );

NETWORK
TITLE = 350 - LCP111_I650_QA1504 - High Temperature Failure - Signal from JUMO

       CALL #"LCP111_I650_QA1504"
       (
         CM_No := 350 ,
         Tab := 28 ,
         SubTab := 7 ,
         CfgType := 0 ,
         CfgInvert := True ,
         InputRaw := LCP111_I650_QA1504_DI_Flt ,
         SC_Local := SL_28_S3 ,
         CM_ALM := #ALM[341] ,
       );

NETWORK
TITLE = 351 - LCP111_N512_BG7501 - Disc Filter 5 Door 1 - Before Filter

       CALL #"LCP111_N512_BG7501"
       (
         CM_No := 351 ,
         Tab := 1 ,
         SubTab := 8 ,
         CfgType := 0 ,
         CfgInvert := True ,
         InputRaw := LCP111_N512_BG7501_DI_ChA ,
         SC_Local := SL_28_S3 ,
         CM_ALM := #ALM[342] ,
       );

NETWORK
TITLE = 352 - LCP111_N512_BG7503 - Disc Filter 5 Door 2 - After Filter

       CALL #"LCP111_N512_BG7503"
       (
         CM_No := 352 ,
         Tab := 1 ,
         SubTab := 8 ,
         CfgType := 0 ,
         CfgInvert := True ,
         InputRaw := LCP111_N512_BG7503_DI_ChA ,
         SC_Local := SL_28_S3 ,
         CM_ALM := #ALM[343] ,
       );

NETWORK
TITLE = 353 - LCP111_N611_BP1525 - Zone 5 Circulation Fan  - Diff. Pressure Circ. Fan 5

       CALL #"LCP111_N611_BP1525"
       (
         CM_No := 353 ,
         Tab := 28 ,
         SubTab := 7 ,
         CfgType := 0 ,
         CfgInvert := True ,
         InputRaw := LCP111_N611_BP1525_DI_Ps ,
         SC_Local := SL_28_S3 ,
         CM_ALM := #ALM[344] ,
       );

NETWORK
TITLE = 354 - LCP111_ES01_SF6559 - Emergency Stop  - Dryer 3 Zone 5 Area

       CALL #"LCP111_ES01_SF6559"
       (
         CM_No := 354 ,
         Tab := 1 ,
         SubTab := 6 ,
         CfgType := 0 ,
         CfgInvert := True ,
         InputRaw := LCP111_ES01_SF6559_DI_ChA ,
         SC_Local := SL_01 ,
         CM_ALM := #ALM[345] ,
       );

NETWORK
TITLE = 355 - LCP111_ES01_SF6560 - Emergency Stop  - LCP111

       CALL #"LCP111_ES01_SF6560"
       (
         CM_No := 355 ,
         Tab := 1 ,
         SubTab := 6 ,
         CfgType := 0 ,
         CfgInvert := True ,
         InputRaw := LCP111_ES01_SF6560_DI_ChA ,
         SC_Local := SL_01 ,
         CM_ALM := #ALM[346] ,
       );

NETWORK
TITLE = 356 - LCP111_DC01_FC1000 - Power Feed Module 24VDC - Status

       CALL #"LCP111_DC01_FC1000"
       (
         CM_No := 356 ,
         Tab := 13 ,
         SubTab := 6 ,
         CfgType := 0 ,
         CfgInvert := True ,
         InputRaw := LCP111_DC01_FC1000_DI_Flt ,
         SC_Local := SL_13 ,
         CM_ALM := #ALM[347] ,
       );

NETWORK
TITLE = 357 - LCP111_IO_KF1000 - Point IO - EtherNet/IP Adapter

       CALL #"LCP111_IO_KF1000"
       (
         CM_No := 357 ,
         Tab := 13 ,
         SubTab := 6 ,
         CfgType := 0 ,
         CfgInvert := True ,
         InputRaw :=  ,
         SC_Local := SL_13 ,
         CM_ALM := #ALM[348] ,
       );

NETWORK
TITLE = 358 - LCP111_IO_KF3013 - 24V DC 8-Point Safety Input Module - SDI

       CALL #"LCP111_IO_KF3013"
       (
         CM_No := 358 ,
         Tab := 13 ,
         SubTab := 6 ,
         CfgType := 0 ,
         CfgInvert := True ,
         InputRaw :=  ,
         SC_Local := SL_13 ,
         CM_ALM := #ALM[349] ,
       );

NETWORK
TITLE = 359 - LCP111_IO_KF3014 - 24V DC 8-Point Safety Input Module - SDI

       CALL #"LCP111_IO_KF3014"
       (
         CM_No := 359 ,
         Tab := 13 ,
         SubTab := 6 ,
         CfgType := 0 ,
         CfgInvert := True ,
         InputRaw :=  ,
         SC_Local := SL_13 ,
         CM_ALM := #ALM[350] ,
       );

NETWORK
TITLE = 360 - LCP112_AC01_FC3601 - 115VAC Power Supply - Thermal Fault

       CALL #"LCP112_AC01_FC3601"
       (
         CM_No := 360 ,
         Tab := 13 ,
         SubTab := 6 ,
         CfgType := 0 ,
         CfgInvert := True ,
         InputRaw := LCP112_AC01_FC3601_DI_Flt ,
         SC_Local := SL_13 ,
         CM_ALM := #ALM[351] ,
       );

NETWORK
TITLE = 361 - LCP112_I660_QA1601 - Min Gas Pressure Switch - (-BP8601)

       CALL #"LCP112_I660_QA1601"
       (
         CM_No := 361 ,
         Tab := 28 ,
         SubTab := 8 ,
         CfgType := 0 ,
         CfgInvert := True ,
         InputRaw := LCP112_I660_QA1601_DI_FltL ,
         SC_Local := SL_28_S3 ,
         CM_ALM := #ALM[352] ,
       );

NETWORK
TITLE = 362 - LCP112_I660_QA1602 - Max Gas Pressure Switch - (-BP8602)

       CALL #"LCP112_I660_QA1602"
       (
         CM_No := 362 ,
         Tab := 28 ,
         SubTab := 8 ,
         CfgType := 0 ,
         CfgInvert := True ,
         InputRaw := LCP112_I660_QA1602_DI_FltH ,
         SC_Local := SL_28_S3 ,
         CM_ALM := #ALM[353] ,
       );

NETWORK
TITLE = 363 - LCP112_I660_QA1603 - Leak Gas Pressure Switch - (-BP8603)

       CALL #"LCP112_I660_QA1603"
       (
         CM_No := 363 ,
         Tab := 28 ,
         SubTab := 8 ,
         CfgType := 0 ,
         CfgInvert := True ,
         InputRaw := LCP112_I660_QA1603_DI_Ps ,
         SC_Local := SL_28_S3 ,
         CM_ALM := #ALM[354] ,
       );

NETWORK
TITLE = 364 - LCP112_I660_QA1613 - No Air Check Pressure Switch - (-BP2613)

       CALL #"LCP112_I660_QA1613"
       (
         CM_No := 364 ,
         Tab := 28 ,
         SubTab := 8 ,
         CfgType := 0 ,
         CfgInvert := True ,
         InputRaw := LCP112_I660_QA1613_DI_Ps ,
         SC_Local := SL_28_S3 ,
         CM_ALM := #ALM[355] ,
       );

NETWORK
TITLE = 365 - LCP112_I660_QA1608 - Burner Failure - Signal from Maxon

       CALL #"LCP112_I660_QA1608"
       (
         CM_No := 365 ,
         Tab := 28 ,
         SubTab := 8 ,
         CfgType := 0 ,
         CfgInvert := True ,
         InputRaw := LCP112_I660_QA1608_DI_Flt ,
         SC_Local := SL_28_S3 ,
         CM_ALM := #ALM[356] ,
       );

NETWORK
TITLE = 366 - LCP112_I660_QA1604 - High Temperature Failure - Signal from JUMO

       CALL #"LCP112_I660_QA1604"
       (
         CM_No := 366 ,
         Tab := 28 ,
         SubTab := 8 ,
         CfgType := 0 ,
         CfgInvert := True ,
         InputRaw := LCP112_I660_QA1604_DI_Flt ,
         SC_Local := SL_28_S3 ,
         CM_ALM := #ALM[357] ,
       );

NETWORK
TITLE = 367 - LCP112_N522_BG7601 - Disc Filter 6 Door 1 - Before Filter

       CALL #"LCP112_N522_BG7601"
       (
         CM_No := 367 ,
         Tab := 1 ,
         SubTab := 8 ,
         CfgType := 0 ,
         CfgInvert := True ,
         InputRaw := LCP112_N522_BG7601_DI_ChA ,
         SC_Local := SL_28_S3 ,
         CM_ALM := #ALM[358] ,
       );

NETWORK
TITLE = 368 - LCP112_N522_BG7603 - Disc Filter 6 Door 2 - After Filter

       CALL #"LCP112_N522_BG7603"
       (
         CM_No := 368 ,
         Tab := 1 ,
         SubTab := 8 ,
         CfgType := 0 ,
         CfgInvert := True ,
         InputRaw := LCP112_N522_BG7603_DI_ChA ,
         SC_Local := SL_28_S3 ,
         CM_ALM := #ALM[359] ,
       );

NETWORK
TITLE = 369 - LCP112_N621_BP1626 - Zone 6 Circulation Fan  - Diff. Pressure Circ. Fan 6

       CALL #"LCP112_N621_BP1626"
       (
         CM_No := 369 ,
         Tab := 28 ,
         SubTab := 8 ,
         CfgType := 0 ,
         CfgInvert := True ,
         InputRaw := LCP112_N621_BP1626_DI_Ps ,
         SC_Local := SL_28_S3 ,
         CM_ALM := #ALM[360] ,
       );

NETWORK
TITLE = 370 - LCP112_ES01_SF6661 - Emergency Stop  - Dryer 3 Zone 6Area

       CALL #"LCP112_ES01_SF6661"
       (
         CM_No := 370 ,
         Tab := 1 ,
         SubTab := 6 ,
         CfgType := 0 ,
         CfgInvert := True ,
         InputRaw := LCP112_ES01_SF6661_DI_ChA ,
         SC_Local := SL_01 ,
         CM_ALM := #ALM[361] ,
       );

NETWORK
TITLE = 371 - LCP112_ES01_SF6662 - Emergency Stop  - LCP112

       CALL #"LCP112_ES01_SF6662"
       (
         CM_No := 371 ,
         Tab := 1 ,
         SubTab := 6 ,
         CfgType := 0 ,
         CfgInvert := True ,
         InputRaw := LCP112_ES01_SF6662_DI_ChA ,
         SC_Local := SL_01 ,
         CM_ALM := #ALM[362] ,
       );

NETWORK
TITLE = 372 - LCP112_DC01_FC1000 - Power Feed Module 24VDC - Status

       CALL #"LCP112_DC01_FC1000"
       (
         CM_No := 372 ,
         Tab := 13 ,
         SubTab := 6 ,
         CfgType := 0 ,
         CfgInvert := True ,
         InputRaw := LCP112_DC01_FC1000_DI_Flt ,
         SC_Local := SL_13 ,
         CM_ALM := #ALM[363] ,
       );

NETWORK
TITLE = 373 - LCP112_IO_KF1000 - Point IO - EtherNet/IP Adapter

       CALL #"LCP112_IO_KF1000"
       (
         CM_No := 373 ,
         Tab := 13 ,
         SubTab := 6 ,
         CfgType := 0 ,
         CfgInvert := True ,
         InputRaw :=  ,
         SC_Local := SL_13 ,
         CM_ALM := #ALM[364] ,
       );

NETWORK
TITLE = 374 - LCP112_IO_KF3013 - 24V DC 8-Point Safety Input Module - SDI

       CALL #"LCP112_IO_KF3013"
       (
         CM_No := 374 ,
         Tab := 13 ,
         SubTab := 6 ,
         CfgType := 0 ,
         CfgInvert := True ,
         InputRaw :=  ,
         SC_Local := SL_13 ,
         CM_ALM := #ALM[365] ,
       );

NETWORK
TITLE = 375 - LCP112_IO_KF3014 - 24V DC 8-Point Safety Input Module - SDI

       CALL #"LCP112_IO_KF3014"
       (
         CM_No := 375 ,
         Tab := 13 ,
         SubTab := 6 ,
         CfgType := 0 ,
         CfgInvert := True ,
         InputRaw :=  ,
         SC_Local := SL_13 ,
         CM_ALM := #ALM[366] ,
       );

NETWORK
TITLE = 376 - LCP113_AC01_FC3701 - 115VAC Power Supply - Thermal Fault

       CALL #"LCP113_AC01_FC3701"
       (
         CM_No := 376 ,
         Tab := 13 ,
         SubTab := 6 ,
         CfgType := 0 ,
         CfgInvert := True ,
         InputRaw := LCP113_AC01_FC3701_DI_Flt ,
         SC_Local := SL_13 ,
         CM_ALM := #ALM[367] ,
       );

NETWORK
TITLE = 377 - LCP113_I670_QA1701 - Min Gas Pressure Switch - (-BP8701)

       CALL #"LCP113_I670_QA1701"
       (
         CM_No := 377 ,
         Tab := 28 ,
         SubTab := 9 ,
         CfgType := 0 ,
         CfgInvert := True ,
         InputRaw := LCP113_I670_QA1701_DI_FltL ,
         SC_Local := SL_28_S3 ,
         CM_ALM := #ALM[368] ,
       );

NETWORK
TITLE = 378 - LCP113_I670_QA1702 - Max Gas Pressure Switch - (-BP8702)

       CALL #"LCP113_I670_QA1702"
       (
         CM_No := 378 ,
         Tab := 28 ,
         SubTab := 9 ,
         CfgType := 0 ,
         CfgInvert := True ,
         InputRaw := LCP113_I670_QA1702_DI_FltH ,
         SC_Local := SL_28_S3 ,
         CM_ALM := #ALM[369] ,
       );

NETWORK
TITLE = 379 - LCP113_I670_QA1703 - Leak Gas Pressure Switch - (-BP8703)

       CALL #"LCP113_I670_QA1703"
       (
         CM_No := 379 ,
         Tab := 28 ,
         SubTab := 9 ,
         CfgType := 0 ,
         CfgInvert := True ,
         InputRaw := LCP113_I670_QA1703_DI_Ps ,
         SC_Local := SL_28_S3 ,
         CM_ALM := #ALM[370] ,
       );

NETWORK
TITLE = 380 - LCP113_I670_QA1713 - No Air Check Pressure Switch - (-BP2713)

       CALL #"LCP113_I670_QA1713"
       (
         CM_No := 380 ,
         Tab := 28 ,
         SubTab := 9 ,
         CfgType := 0 ,
         CfgInvert := True ,
         InputRaw := LCP113_I670_QA1713_DI_Ps ,
         SC_Local := SL_28_S3 ,
         CM_ALM := #ALM[371] ,
       );

NETWORK
TITLE = 381 - LCP113_I670_QA1708 - Burner Failure - Signal from Maxon

       CALL #"LCP113_I670_QA1708"
       (
         CM_No := 381 ,
         Tab := 28 ,
         SubTab := 9 ,
         CfgType := 0 ,
         CfgInvert := True ,
         InputRaw := LCP113_I670_QA1708_DI_Flt ,
         SC_Local := SL_28_S3 ,
         CM_ALM := #ALM[372] ,
       );

NETWORK
TITLE = 382 - LCP113_I670_QA1704 - High Temperature Failure - Signal from JUMO

       CALL #"LCP113_I670_QA1704"
       (
         CM_No := 382 ,
         Tab := 28 ,
         SubTab := 9 ,
         CfgType := 0 ,
         CfgInvert := True ,
         InputRaw := LCP113_I670_QA1704_DI_Flt ,
         SC_Local := SL_28_S3 ,
         CM_ALM := #ALM[373] ,
       );

NETWORK
TITLE = 383 - LCP113_N532_BG7701 - Disc Filter 7 Door 1 - Before Filter

       CALL #"LCP113_N532_BG7701"
       (
         CM_No := 383 ,
         Tab := 1 ,
         SubTab := 8 ,
         CfgType := 0 ,
         CfgInvert := True ,
         InputRaw := LCP113_N532_BG7701_DI_ChA ,
         SC_Local := SL_28_S3 ,
         CM_ALM := #ALM[374] ,
       );

NETWORK
TITLE = 384 - LCP113_N532_BG7703 - Disc Filter 7 Door 2 - After Filter

       CALL #"LCP113_N532_BG7703"
       (
         CM_No := 384 ,
         Tab := 1 ,
         SubTab := 8 ,
         CfgType := 0 ,
         CfgInvert := True ,
         InputRaw := LCP113_N532_BG7703_DI_ChA ,
         SC_Local := SL_28_S3 ,
         CM_ALM := #ALM[375] ,
       );

NETWORK
TITLE = 385 - LCP113_N631_BP1727 - Zone 7 Circulation Fan - Diff. Pressure Circ. Fan 7

       CALL #"LCP113_N631_BP1727"
       (
         CM_No := 385 ,
         Tab := 28 ,
         SubTab := 9 ,
         CfgType := 0 ,
         CfgInvert := True ,
         InputRaw := LCP113_N631_BP1727_DI_Ps ,
         SC_Local := SL_28_S3 ,
         CM_ALM := #ALM[376] ,
       );

NETWORK
TITLE = 386 - LCP113_ES01_SF6762 - Emergency Stop  - Dryer 3 Zone 7 Area

       CALL #"LCP113_ES01_SF6762"
       (
         CM_No := 386 ,
         Tab := 1 ,
         SubTab := 6 ,
         CfgType := 0 ,
         CfgInvert := True ,
         InputRaw := LCP113_ES01_SF6762_DI_ChA ,
         SC_Local := SL_01 ,
         CM_ALM := #ALM[377] ,
       );

NETWORK
TITLE = 387 - LCP113_ES01_SF6763 - Emergency Stop  - LCP113

       CALL #"LCP113_ES01_SF6763"
       (
         CM_No := 387 ,
         Tab := 1 ,
         SubTab := 6 ,
         CfgType := 0 ,
         CfgInvert := True ,
         InputRaw := LCP113_ES01_SF6763_DI_ChA ,
         SC_Local := SL_01 ,
         CM_ALM := #ALM[378] ,
       );

NETWORK
TITLE = 388 - LCP113_DC01_FC1000 - Power Feed Module 24VDC - Status

       CALL #"LCP113_DC01_FC1000"
       (
         CM_No := 388 ,
         Tab := 13 ,
         SubTab := 6 ,
         CfgType := 0 ,
         CfgInvert := True ,
         InputRaw := LCP113_DC01_FC1000_DI_Flt ,
         SC_Local := SL_13 ,
         CM_ALM := #ALM[379] ,
       );

NETWORK
TITLE = 389 - LCP113_IO_KF1000 - Point IO - EtherNet/IP Adapter

       CALL #"LCP113_IO_KF1000"
       (
         CM_No := 389 ,
         Tab := 13 ,
         SubTab := 6 ,
         CfgType := 0 ,
         CfgInvert := True ,
         InputRaw :=  ,
         SC_Local := SL_13 ,
         CM_ALM := #ALM[380] ,
       );

NETWORK
TITLE = 390 - LCP113_IO_KF3013 - 24V DC 8-Point Safety Input Module - SDI

       CALL #"LCP113_IO_KF3013"
       (
         CM_No := 390 ,
         Tab := 13 ,
         SubTab := 6 ,
         CfgType := 0 ,
         CfgInvert := True ,
         InputRaw :=  ,
         SC_Local := SL_13 ,
         CM_ALM := #ALM[381] ,
       );

NETWORK
TITLE = 391 - LCP113_IO_KF3014 - 24V DC 8-Point Safety Input Module - SDI

       CALL #"LCP113_IO_KF3014"
       (
         CM_No := 391 ,
         Tab := 13 ,
         SubTab := 6 ,
         CfgType := 0 ,
         CfgInvert := True ,
         InputRaw :=  ,
         SC_Local := SL_13 ,
         CM_ALM := #ALM[382] ,
       );

NETWORK
TITLE = 392 - LCP121_ES01_SF6181 - Emergency Stop  - CB.121-01

       CALL #"LCP121_ES01_SF6181"
       (
         CM_No := 392 ,
         Tab := 1 ,
         SubTab := 7 ,
         CfgType := 0 ,
         CfgInvert := True ,
         InputRaw := LCP121_ES01_SF6181_DI_ChA ,
         SC_Local := SL_01 ,
         CM_ALM := #ALM[383] ,
       );

NETWORK
TITLE = 393 - LCP121_ES01_SF6182 - Emergency Stop  - CB.121-02

       CALL #"LCP121_ES01_SF6182"
       (
         CM_No := 393 ,
         Tab := 1 ,
         SubTab := 7 ,
         CfgType := 0 ,
         CfgInvert := True ,
         InputRaw := LCP121_ES01_SF6182_DI_ChA ,
         SC_Local := SL_01 ,
         CM_ALM := #ALM[384] ,
       );

NETWORK
TITLE = 394 - LCP121_DC01_FC1000 - Power Feed Module 24VDC - Status

       CALL #"LCP121_DC01_FC1000"
       (
         CM_No := 394 ,
         Tab := 13 ,
         SubTab := 7 ,
         CfgType := 0 ,
         CfgInvert := True ,
         InputRaw := LCP121_DC01_FC1000_DI_Flt ,
         SC_Local := SL_13 ,
         CM_ALM := #ALM[385] ,
       );

NETWORK
TITLE = 395 - LCP122_ES01_SF6184 - Emergency Stop  - CB122-01

       CALL #"LCP122_ES01_SF6184"
       (
         CM_No := 395 ,
         Tab := 1 ,
         SubTab := 7 ,
         CfgType := 0 ,
         CfgInvert := True ,
         InputRaw := LCP122_ES01_SF6184_DI_ChA ,
         SC_Local := SL_01 ,
         CM_ALM := #ALM[386] ,
       );

NETWORK
TITLE = 396 - LCP122_ES01_SF6185 - Emergency Stop  - CB122-02

       CALL #"LCP122_ES01_SF6185"
       (
         CM_No := 396 ,
         Tab := 1 ,
         SubTab := 7 ,
         CfgType := 0 ,
         CfgInvert := True ,
         InputRaw := LCP122_ES01_SF6185_DI_ChA ,
         SC_Local := SL_01 ,
         CM_ALM := #ALM[387] ,
       );

NETWORK
TITLE = 397 - LCP122_ES01_SF6186 - Emergency Stop  - CB.122-03

       CALL #"LCP122_ES01_SF6186"
       (
         CM_No := 397 ,
         Tab := 1 ,
         SubTab := 7 ,
         CfgType := 0 ,
         CfgInvert := True ,
         InputRaw := LCP122_ES01_SF6186_DI_ChA ,
         SC_Local := SL_01 ,
         CM_ALM := #ALM[388] ,
       );

NETWORK
TITLE = 398 - LCP122_DC01_FC1000 - Power Feed Module 24VDC - Status

       CALL #"LCP122_DC01_FC1000"
       (
         CM_No := 398 ,
         Tab := 13 ,
         SubTab := 7 ,
         CfgType := 0 ,
         CfgInvert := True ,
         InputRaw := LCP122_DC01_FC1000_DI_Flt ,
         SC_Local := SL_13 ,
         CM_ALM := #ALM[389] ,
       );

NETWORK
TITLE = 399 - LCP123_ES01_SF6188 - Emergency Stop  - CB.123-01

       CALL #"LCP123_ES01_SF6188"
       (
         CM_No := 399 ,
         Tab := 1 ,
         SubTab := 7 ,
         CfgType := 0 ,
         CfgInvert := True ,
         InputRaw := LCP123_ES01_SF6188_DI_ChA ,
         SC_Local := SL_01 ,
         CM_ALM := #ALM[390] ,
       );

NETWORK
TITLE = 400 - LCP122_ES01_SF6190 - Emergency Stop  - CB.122-04

       CALL #"LCP122_ES01_SF6190"
       (
         CM_No := 400 ,
         Tab := 1 ,
         SubTab := 7 ,
         CfgType := 0 ,
         CfgInvert := True ,
         InputRaw := LCP122_ES01_SF6190_DI_ChA ,
         SC_Local := SL_01 ,
         CM_ALM := #ALM[391] ,
       );

NETWORK
TITLE = 401 - LCP123_DC01_FC1000 - Power Feed Module 24VDC - Status

       CALL #"LCP123_DC01_FC1000"
       (
         CM_No := 401 ,
         Tab := 13 ,
         SubTab := 7 ,
         CfgType := 0 ,
         CfgInvert := True ,
         InputRaw := LCP123_DC01_FC1000_DI_Flt ,
         SC_Local := SL_13 ,
         CM_ALM := #ALM[392] ,
       );

NETWORK
TITLE = 402 - LCP121_IO_KF1000 - Point IO - EtherNet/IP Adapter

       CALL #"LCP121_IO_KF1000"
       (
         CM_No := 402 ,
         Tab := 13 ,
         SubTab := 5 ,
         CfgType := 0 ,
         CfgInvert := True ,
         InputRaw :=  ,
         SC_Local := SL_13 ,
         CM_ALM := #ALM[393] ,
       );

NETWORK
TITLE = 403 - LCP121_IO_KF3010 - 24V DC 8-Point Safety Input Module - SDI

       CALL #"LCP121_IO_KF3010"
       (
         CM_No := 403 ,
         Tab := 13 ,
         SubTab := 5 ,
         CfgType := 0 ,
         CfgInvert := True ,
         InputRaw :=  ,
         SC_Local := SL_13 ,
         CM_ALM := #ALM[394] ,
       );

NETWORK
TITLE = 404 - LCP131_I811_BP1201 - Zone 1 Burner Fan - Differential Pressure Sensor

       CALL #"LCP131_I811_BP1201"
       (
         CM_No := 404 ,
         Tab := 28 ,
         SubTab := 3 ,
         CfgType := 0 ,
         CfgInvert := True ,
         InputRaw := LCP131_I811_BP1201_DI_Ps ,
         SC_Local := SL_28_S1 ,
         CM_ALM := #ALM[395] ,
       );

NETWORK
TITLE = 405 - LCP131_K811_BP1202 - Zone 3 Burner Fan - Differential Pressure Sensor

       CALL #"LCP131_K811_BP1202"
       (
         CM_No := 405 ,
         Tab := 28 ,
         SubTab := 5 ,
         CfgType := 0 ,
         CfgInvert := True ,
         InputRaw := LCP131_K811_BP1202_DI_Ps ,
         SC_Local := SL_28_S2 ,
         CM_ALM := #ALM[396] ,
       );

NETWORK
TITLE = 406 - LCP131_K821_BP1203 - Zone 4 Burner Fan - Differential Pressure Sensor

       CALL #"LCP131_K821_BP1203"
       (
         CM_No := 406 ,
         Tab := 28 ,
         SubTab := 6 ,
         CfgType := 0 ,
         CfgInvert := True ,
         InputRaw := LCP131_K821_BP1203_DI_Ps ,
         SC_Local := SL_28_S2 ,
         CM_ALM := #ALM[397] ,
       );

NETWORK
TITLE = 407 - LCP131_N811_BP1204 - Zone 5 Burner Fan - Differential Pressure Sensor

       CALL #"LCP131_N811_BP1204"
       (
         CM_No := 407 ,
         Tab := 28 ,
         SubTab := 7 ,
         CfgType := 0 ,
         CfgInvert := True ,
         InputRaw := LCP131_N811_BP1204_DI_Ps ,
         SC_Local := SL_28_S3 ,
         CM_ALM := #ALM[398] ,
       );

NETWORK
TITLE = 408 - LCP131_N821_BP1205 - Zone 6 Burner Fan - Differential Pressure Sensor

       CALL #"LCP131_N821_BP1205"
       (
         CM_No := 408 ,
         Tab := 28 ,
         SubTab := 8 ,
         CfgType := 0 ,
         CfgInvert := True ,
         InputRaw := LCP131_N821_BP1205_DI_Ps ,
         SC_Local := SL_28_S3 ,
         CM_ALM := #ALM[399] ,
       );

NETWORK
TITLE = 409 - LCP131_N831_BP1206 - Zone 7 Burner Fan - Differential Pressure Sensor

       CALL #"LCP131_N831_BP1206"
       (
         CM_No := 409 ,
         Tab := 28 ,
         SubTab := 9 ,
         CfgType := 0 ,
         CfgInvert := True ,
         InputRaw := LCP131_N831_BP1206_DI_Ps ,
         SC_Local := SL_28_S3 ,
         CM_ALM := #ALM[400] ,
       );

NETWORK
TITLE = 410 - LCP131_I711_BP1207 - Exhaust Fan 1 - Differential Pressure Sensor

       CALL #"LCP131_I711_BP1207"
       (
         CM_No := 410 ,
         Tab := 28 ,
         SubTab := 3 ,
         CfgType := 0 ,
         CfgInvert := True ,
         InputRaw := LCP131_I711_BP1207_DI_Ps ,
         SC_Local := SL_28_S1 ,
         CM_ALM := #ALM[401] ,
       );

NETWORK
TITLE = 411 - LCP131_K711_BP1208 - Exhaust Fan 3 - Differential Pressure Sensor

       CALL #"LCP131_K711_BP1208"
       (
         CM_No := 411 ,
         Tab := 28 ,
         SubTab := 5 ,
         CfgType := 0 ,
         CfgInvert := True ,
         InputRaw := LCP131_K711_BP1208_DI_Ps ,
         SC_Local := SL_28_S2 ,
         CM_ALM := #ALM[402] ,
       );

NETWORK
TITLE = 412 - LCP131_K721_BP1209 - Exhaust Fan 4 - Differential Pressure Sensor

       CALL #"LCP131_K721_BP1209"
       (
         CM_No := 412 ,
         Tab := 28 ,
         SubTab := 6 ,
         CfgType := 0 ,
         CfgInvert := True ,
         InputRaw := LCP131_K721_BP1209_DI_Ps ,
         SC_Local := SL_28_S2 ,
         CM_ALM := #ALM[403] ,
       );

NETWORK
TITLE = 413 - LCP131_N711_BP1210 - Exhaust Fan 5 - Differential Pressure Sensor

       CALL #"LCP131_N711_BP1210"
       (
         CM_No := 413 ,
         Tab := 28 ,
         SubTab := 7 ,
         CfgType := 0 ,
         CfgInvert := True ,
         InputRaw := LCP131_N711_BP1210_DI_Ps ,
         SC_Local := SL_28_S3 ,
         CM_ALM := #ALM[404] ,
       );

NETWORK
TITLE = 414 - LCP131_N721_BP1211 - Exhaust Fan 6 - Differential Pressure Sensor

       CALL #"LCP131_N721_BP1211"
       (
         CM_No := 414 ,
         Tab := 28 ,
         SubTab := 8 ,
         CfgType := 0 ,
         CfgInvert := True ,
         InputRaw := LCP131_N721_BP1211_DI_Ps ,
         SC_Local := SL_28_S3 ,
         CM_ALM := #ALM[405] ,
       );

NETWORK
TITLE = 415 - LCP131_N731_BP1212 - Exhaust Fan 7 - Differential Pressure Sensor

       CALL #"LCP131_N731_BP1212"
       (
         CM_No := 415 ,
         Tab := 28 ,
         SubTab := 9 ,
         CfgType := 0 ,
         CfgInvert := True ,
         InputRaw := LCP131_N731_BP1212_DI_Ps ,
         SC_Local := SL_28_S3 ,
         CM_ALM := #ALM[406] ,
       );

NETWORK
TITLE = 416 - LCP131_ES01_SF6191 - Emergency Stop  - Fan Area

       CALL #"LCP131_ES01_SF6191"
       (
         CM_No := 416 ,
         Tab := 1 ,
         SubTab := 6 ,
         CfgType := 0 ,
         CfgInvert := True ,
         InputRaw := LCP131_ES01_SF6191_DI_ChA ,
         SC_Local := SL_01 ,
         CM_ALM := #ALM[407] ,
       );

NETWORK
TITLE = 417 - LCP131_ES01_SF6192 - Emergency Stop  - Fan Area

       CALL #"LCP131_ES01_SF6192"
       (
         CM_No := 417 ,
         Tab := 1 ,
         SubTab := 6 ,
         CfgType := 0 ,
         CfgInvert := True ,
         InputRaw := LCP131_ES01_SF6192_DI_ChA ,
         SC_Local := SL_01 ,
         CM_ALM := #ALM[408] ,
       );

NETWORK
TITLE = 418 - LCP131_ES01_SF6193 - Emergency Stop  - Fan Area

       CALL #"LCP131_ES01_SF6193"
       (
         CM_No := 418 ,
         Tab := 1 ,
         SubTab := 6 ,
         CfgType := 0 ,
         CfgInvert := True ,
         InputRaw := LCP131_ES01_SF6193_DI_ChA ,
         SC_Local := SL_01 ,
         CM_ALM := #ALM[409] ,
       );

NETWORK
TITLE = 419 - LCP131_ES01_SF6194 - Emergency Stop  - LCP131

       CALL #"LCP131_ES01_SF6194"
       (
         CM_No := 419 ,
         Tab := 1 ,
         SubTab := 6 ,
         CfgType := 0 ,
         CfgInvert := True ,
         InputRaw := LCP131_ES01_SF6194_DI_ChA ,
         SC_Local := SL_01 ,
         CM_ALM := #ALM[410] ,
       );

NETWORK
TITLE = 420 - LCP131_DC01_FC1000 - Power Feed Module 24VDC - Status

       CALL #"LCP131_DC01_FC1000"
       (
         CM_No := 420 ,
         Tab := 13 ,
         SubTab := 7 ,
         CfgType := 0 ,
         CfgInvert := True ,
         InputRaw := LCP131_DC01_FC1000_DI_Flt ,
         SC_Local := SL_13 ,
         CM_ALM := #ALM[411] ,
       );

NETWORK
TITLE = 421 - LCP131_IO_KF1000 - Point IO - EtherNet/IP Adapter

       CALL #"LCP131_IO_KF1000"
       (
         CM_No := 421 ,
         Tab := 13 ,
         SubTab := 5 ,
         CfgType := 0 ,
         CfgInvert := True ,
         InputRaw :=  ,
         SC_Local := SL_13 ,
         CM_ALM := #ALM[412] ,
       );

NETWORK
TITLE = 422 - LCP131_IO_KF3012 - 24V DC 8-Point Safety Input Module - SDI

       CALL #"LCP131_IO_KF3012"
       (
         CM_No := 422 ,
         Tab := 13 ,
         SubTab := 5 ,
         CfgType := 0 ,
         CfgInvert := True ,
         InputRaw :=  ,
         SC_Local := SL_13 ,
         CM_ALM := #ALM[413] ,
       );

NETWORK
TITLE = 423 - LCP131_IO_KF3013 - 24V DC 8-Point Safety Input Module - SDI

       CALL #"LCP131_IO_KF3013"
       (
         CM_No := 423 ,
         Tab := 13 ,
         SubTab := 5 ,
         CfgType := 0 ,
         CfgInvert := True ,
         InputRaw :=  ,
         SC_Local := SL_13 ,
         CM_ALM := #ALM[414] ,
       );

NETWORK
TITLE = 424 - LCP131_IO_KF3014 - 24V DC 8-Point Safety Input Module - SDI

       CALL #"LCP131_IO_KF3014"
       (
         CM_No := 424 ,
         Tab := 13 ,
         SubTab := 5 ,
         CfgType := 0 ,
         CfgInvert := True ,
         InputRaw :=  ,
         SC_Local := SL_13 ,
         CM_ALM := #ALM[415] ,
       );

NETWORK
TITLE = 425 - LCP132_Q710_BG7502 - Mixing Tank - Inspection Hatch - Safety Switch

       CALL #"LCP132_Q710_BG7502"
       (
         CM_No := 425 ,
         Tab := 29 ,
         SubTab := 2 ,
         CfgType := 0 ,
         CfgInvert := True ,
         InputRaw := LCP132_Q710_BG7502_DI_ChA ,
         SC_Local := SL_29_P ,
         CM_ALM := #ALM[416] ,
       );

NETWORK
TITLE = 426 - LCP132_ES01_SF6164 - Emergency Stop  - LCP132

       CALL #"LCP132_ES01_SF6164"
       (
         CM_No := 426 ,
         Tab := 1 ,
         SubTab := 7 ,
         CfgType := 0 ,
         CfgInvert := True ,
         InputRaw := LCP132_ES01_SF6164_DI_ChA ,
         SC_Local := SL_01 ,
         CM_ALM := #ALM[417] ,
       );

NETWORK
TITLE = 427 - LCP132_DC01_FC1000 - Power Feed Module 24VDC - Status

       CALL #"LCP132_DC01_FC1000"
       (
         CM_No := 427 ,
         Tab := 13 ,
         SubTab := 7 ,
         CfgType := 0 ,
         CfgInvert := True ,
         InputRaw := LCP132_DC01_FC1000_DI_Flt ,
         SC_Local := SL_13 ,
         CM_ALM := #ALM[418] ,
       );

NETWORK
TITLE = 428 - PLC1.1_AC01_FC2010 - 115VAC Power Supply - Circuit Breaker

       CALL #"PLC1.1_AC01_FC2010"
       (
         CM_No := 428 ,
         Tab := 13 ,
         SubTab := 1 ,
         CfgType := 0 ,
         CfgInvert := True ,
         InputRaw := PLC1_AC01_FC2010_DI_Flt ,
         SC_Local := SL_13 ,
         CM_ALM := #ALM[419] ,
       );

NETWORK
TITLE = 429 - PLC1.1_AC01_FC1791 - Power Supply 115VAC LCP101 - Burner 1

       CALL #"PLC1.1_AC01_FC1791"
       (
         CM_No := 429 ,
         Tab := 13 ,
         SubTab := 2 ,
         CfgType := 0 ,
         CfgInvert := True ,
         InputRaw := PLC1_AC01_FC1791_DI_Flt ,
         SC_Local := SL_13 ,
         CM_ALM := #ALM[420] ,
       );

NETWORK
TITLE = 430 - PLC1.1_AC02_FC2011 - 115VAC Power Supply - Circuit Breaker

       CALL #"PLC1.1_AC02_FC2011"
       (
         CM_No := 430 ,
         Tab := 13 ,
         SubTab := 1 ,
         CfgType := 0 ,
         CfgInvert := True ,
         InputRaw := PLC1_AC02_FC2011_DI_Flt ,
         SC_Local := SL_13 ,
         CM_ALM := #ALM[421] ,
       );

NETWORK
TITLE = 431 - PLC1.1_AC02_FC1792 - Power Supply 115VAC LCP102 - Burner 2

       CALL #"PLC1.1_AC02_FC1792"
       (
         CM_No := 431 ,
         Tab := 13 ,
         SubTab := 2 ,
         CfgType := 0 ,
         CfgInvert := True ,
         InputRaw := PLC1_AC02_FC1792_DI_Flt ,
         SC_Local := SL_13 ,
         CM_ALM := #ALM[422] ,
       );

NETWORK
TITLE = 432 - PLC1.1_AC02_FC1793 - Power Supply 115VAC LCP103 - Burner 3

       CALL #"PLC1.1_AC02_FC1793"
       (
         CM_No := 432 ,
         Tab := 13 ,
         SubTab := 2 ,
         CfgType := 0 ,
         CfgInvert := True ,
         InputRaw := PLC1_AC02_FC1793_DI_Flt ,
         SC_Local := SL_13 ,
         CM_ALM := #ALM[423] ,
       );

NETWORK
TITLE = 433 - PLC1.1_AC03_FC2012 - 115VAC Power Supply - Circuit Breaker

       CALL #"PLC1.1_AC03_FC2012"
       (
         CM_No := 433 ,
         Tab := 13 ,
         SubTab := 1 ,
         CfgType := 0 ,
         CfgInvert := True ,
         InputRaw := PLC1_AC03_FC2012_DI_Flt ,
         SC_Local := SL_13 ,
         CM_ALM := #ALM[424] ,
       );

NETWORK
TITLE = 434 - PLC1.1_AC03_FC1794 - Power Supply 115VAC LCP104 - Burner 4

       CALL #"PLC1.1_AC03_FC1794"
       (
         CM_No := 434 ,
         Tab := 13 ,
         SubTab := 2 ,
         CfgType := 0 ,
         CfgInvert := True ,
         InputRaw := PLC1_AC03_FC1794_DI_Flt ,
         SC_Local := SL_13 ,
         CM_ALM := #ALM[425] ,
       );

NETWORK
TITLE = 435 - PLC1.1_AC03_FC1795 - Power Supply 115VAC LCP111 - Burner 5

       CALL #"PLC1.1_AC03_FC1795"
       (
         CM_No := 435 ,
         Tab := 13 ,
         SubTab := 2 ,
         CfgType := 0 ,
         CfgInvert := True ,
         InputRaw := PLC1_AC03_FC1795_DI_Flt ,
         SC_Local := SL_13 ,
         CM_ALM := #ALM[426] ,
       );

NETWORK
TITLE = 436 - PLC1.1_AC04_FC2013 - 115VAC Power Supply - Circuit Breaker

       CALL #"PLC1.1_AC04_FC2013"
       (
         CM_No := 436 ,
         Tab := 13 ,
         SubTab := 1 ,
         CfgType := 0 ,
         CfgInvert := True ,
         InputRaw := PLC1_AC04_FC2013_DI_Flt ,
         SC_Local := SL_13 ,
         CM_ALM := #ALM[427] ,
       );

NETWORK
TITLE = 437 - PLC1.1_AC04_FC1796 - Power Supply 115VAC LCP112 - Burner 6

       CALL #"PLC1.1_AC04_FC1796"
       (
         CM_No := 437 ,
         Tab := 13 ,
         SubTab := 2 ,
         CfgType := 0 ,
         CfgInvert := True ,
         InputRaw := PLC1_AC04_FC1796_DI_Flt ,
         SC_Local := SL_13 ,
         CM_ALM := #ALM[428] ,
       );

NETWORK
TITLE = 438 - PLC1.1_AC04_FC1797 - Power Supply 115VAC LCP113 - Burner 7

       CALL #"PLC1.1_AC04_FC1797"
       (
         CM_No := 438 ,
         Tab := 13 ,
         SubTab := 2 ,
         CfgType := 0 ,
         CfgInvert := True ,
         InputRaw := PLC1_AC04_FC1797_DI_Flt ,
         SC_Local := SL_13 ,
         CM_ALM := #ALM[429] ,
       );

NETWORK
TITLE = 439 - PLC1.1_DC01_FC1010 - Power Feed Module 24VDC - Status

       CALL #"PLC1.1_DC01_FC1010"
       (
         CM_No := 439 ,
         Tab := 13 ,
         SubTab := 1 ,
         CfgType := 0 ,
         CfgInvert := True ,
         InputRaw := PLC1_DC01_FC1010_DI_Sts ,
         SC_Local := SL_13 ,
         CM_ALM := #ALM[430] ,
       );

NETWORK
TITLE = 440 - PLC1.1_DC02_1LDC1L - Power Supply 24VDC - MCC10

       CALL #"PLC1.1_DC02_1LDC1L"
       (
         CM_No := 440 ,
         Tab := 13 ,
         SubTab := 1 ,
         CfgType := 0 ,
         CfgInvert := True ,
         InputRaw := PLC1_DC02_1LDC1L_DI_Flt ,
         SC_Local := SL_13 ,
         CM_ALM := #ALM[431] ,
       );

NETWORK
TITLE = 441 - PLC1.1_DC02_2LDC2L - Power Supply 24VDC - LCP101

       CALL #"PLC1.1_DC02_2LDC2L"
       (
         CM_No := 441 ,
         Tab := 13 ,
         SubTab := 1 ,
         CfgType := 0 ,
         CfgInvert := True ,
         InputRaw := PLC1_DC02_2LDC2L_DI_Flt ,
         SC_Local := SL_13 ,
         CM_ALM := #ALM[432] ,
       );

NETWORK
TITLE = 442 - PLC1.1_DC02_3LDC3L - Power Supply 24VDC - LCP102

       CALL #"PLC1.1_DC02_3LDC3L"
       (
         CM_No := 442 ,
         Tab := 13 ,
         SubTab := 1 ,
         CfgType := 0 ,
         CfgInvert := True ,
         InputRaw := PLC1_DC02_3LDC3L_DI_Flt ,
         SC_Local := SL_13 ,
         CM_ALM := #ALM[433] ,
       );

NETWORK
TITLE = 443 - PLC1.1_DC03_1LDC1L - Power Supply 24VDC - LCP103

       CALL #"PLC1.1_DC03_1LDC1L"
       (
         CM_No := 443 ,
         Tab := 13 ,
         SubTab := 1 ,
         CfgType := 0 ,
         CfgInvert := True ,
         InputRaw := PLC1_DC03_1LDC1L_DI_Flt ,
         SC_Local := SL_13 ,
         CM_ALM := #ALM[434] ,
       );

NETWORK
TITLE = 444 - PLC1.1_DC03_2LDC2L - Power Supply 24VDC - LCP104

       CALL #"PLC1.1_DC03_2LDC2L"
       (
         CM_No := 444 ,
         Tab := 13 ,
         SubTab := 1 ,
         CfgType := 0 ,
         CfgInvert := True ,
         InputRaw := PLC1_DC03_2LDC2L_DI_Flt ,
         SC_Local := SL_13 ,
         CM_ALM := #ALM[435] ,
       );

NETWORK
TITLE = 445 - PLC1.1_DC03_3LDC3L - Power Supply 24VDC - Spare

       CALL #"PLC1.1_DC03_3LDC3L"
       (
         CM_No := 445 ,
         Tab := 13 ,
         SubTab := 1 ,
         CfgType := 0 ,
         CfgInvert := True ,
         InputRaw := PLC1_DC03_3LDC3L_DI_Flt ,
         SC_Local := SL_13 ,
         CM_ALM := #ALM[436] ,
       );

NETWORK
TITLE = 446 - PLC1.1_DC04_1LDC1L - Power Supply 24VDC - MCC11

       CALL #"PLC1.1_DC04_1LDC1L"
       (
         CM_No := 446 ,
         Tab := 13 ,
         SubTab := 1 ,
         CfgType := 0 ,
         CfgInvert := True ,
         InputRaw := PLC1_DC04_1LDC1L_DI_Flt ,
         SC_Local := SL_13 ,
         CM_ALM := #ALM[437] ,
       );

NETWORK
TITLE = 447 - PLC1.1_DC04_2LDC2L - Power Supply 24VDC - LCP111

       CALL #"PLC1.1_DC04_2LDC2L"
       (
         CM_No := 447 ,
         Tab := 13 ,
         SubTab := 1 ,
         CfgType := 0 ,
         CfgInvert := True ,
         InputRaw := PLC1_DC04_2LDC2L_DI_Flt ,
         SC_Local := SL_13 ,
         CM_ALM := #ALM[438] ,
       );

NETWORK
TITLE = 448 - PLC1.1_DC04_3LDC3L - Power Supply 24VDC - LCP112

       CALL #"PLC1.1_DC04_3LDC3L"
       (
         CM_No := 448 ,
         Tab := 13 ,
         SubTab := 1 ,
         CfgType := 0 ,
         CfgInvert := True ,
         InputRaw := PLC1_DC04_3LDC3L_DI_Flt ,
         SC_Local := SL_13 ,
         CM_ALM := #ALM[439] ,
       );

NETWORK
TITLE = 449 - PLC1.1_DC04_4LDC4L - Power Supply 24VDC - LCP113

       CALL #"PLC1.1_DC04_4LDC4L"
       (
         CM_No := 449 ,
         Tab := 13 ,
         SubTab := 1 ,
         CfgType := 0 ,
         CfgInvert := True ,
         InputRaw := PLC1_DC04_4LDC4L_DI_Flt ,
         SC_Local := SL_13 ,
         CM_ALM := #ALM[440] ,
       );

NETWORK
TITLE = 450 - PLC1.1_DC05_1LDC1L - Power Supply 24VDC - MCC12

       CALL #"PLC1.1_DC05_1LDC1L"
       (
         CM_No := 450 ,
         Tab := 13 ,
         SubTab := 1 ,
         CfgType := 0 ,
         CfgInvert := True ,
         InputRaw := PLC1_DC05_1LDC1L_DI_Flt ,
         SC_Local := SL_13 ,
         CM_ALM := #ALM[441] ,
       );

NETWORK
TITLE = 451 - PLC1.1_DC05_2LDC2L - Power Supply 24VDC - LCP121

       CALL #"PLC1.1_DC05_2LDC2L"
       (
         CM_No := 451 ,
         Tab := 13 ,
         SubTab := 1 ,
         CfgType := 0 ,
         CfgInvert := True ,
         InputRaw := PLC1_DC05_2LDC2L_DI_Flt ,
         SC_Local := SL_13 ,
         CM_ALM := #ALM[442] ,
       );

NETWORK
TITLE = 452 - PLC1.1_DC05_3LDC3L - Power Supply 24VDC - LCP122

       CALL #"PLC1.1_DC05_3LDC3L"
       (
         CM_No := 452 ,
         Tab := 13 ,
         SubTab := 1 ,
         CfgType := 0 ,
         CfgInvert := True ,
         InputRaw := PLC1_DC05_3LDC3L_DI_Flt ,
         SC_Local := SL_13 ,
         CM_ALM := #ALM[443] ,
       );

NETWORK
TITLE = 453 - PLC1.1_DC05_4LDC4L - Power Supply 24VDC - LCP123

       CALL #"PLC1.1_DC05_4LDC4L"
       (
         CM_No := 453 ,
         Tab := 13 ,
         SubTab := 1 ,
         CfgType := 0 ,
         CfgInvert := True ,
         InputRaw := PLC1_DC05_4LDC4L_DI_Flt ,
         SC_Local := SL_13 ,
         CM_ALM := #ALM[444] ,
       );

NETWORK
TITLE = 454 - PLC1.1_DC06_1LDC1L - Power Supply 24VDC - MCC13

       CALL #"PLC1.1_DC06_1LDC1L"
       (
         CM_No := 454 ,
         Tab := 13 ,
         SubTab := 1 ,
         CfgType := 0 ,
         CfgInvert := True ,
         InputRaw := PLC1_DC06_1LDC1L_DI_Flt ,
         SC_Local := SL_13 ,
         CM_ALM := #ALM[445] ,
       );

NETWORK
TITLE = 455 - PLC1.1_DC06_2LDC2L - Power Supply 24VDC - LCP131

       CALL #"PLC1.1_DC06_2LDC2L"
       (
         CM_No := 455 ,
         Tab := 13 ,
         SubTab := 1 ,
         CfgType := 0 ,
         CfgInvert := True ,
         InputRaw := PLC1_DC06_2LDC2L_DI_Flt ,
         SC_Local := SL_13 ,
         CM_ALM := #ALM[446] ,
       );

NETWORK
TITLE = 456 - PLC1.1_DC06_3LDC3L - Power Supply 24VDC - LCP132

       CALL #"PLC1.1_DC06_3LDC3L"
       (
         CM_No := 456 ,
         Tab := 13 ,
         SubTab := 1 ,
         CfgType := 0 ,
         CfgInvert := True ,
         InputRaw := PLC1_DC06_3LDC3L_DI_Flt ,
         SC_Local := SL_13 ,
         CM_ALM := #ALM[447] ,
       );

NETWORK
TITLE = 457 - PLC1.1_DC06_4LDC4L - Power Supply 24VDC - Spare

       CALL #"PLC1.1_DC06_4LDC4L"
       (
         CM_No := 457 ,
         Tab := 13 ,
         SubTab := 1 ,
         CfgType := 0 ,
         CfgInvert := True ,
         InputRaw := PLC1_DC06_4LDC4L_DI_Flt ,
         SC_Local := SL_13 ,
         CM_ALM := #ALM[448] ,
       );

NETWORK
TITLE = 458 - PLC1.1_DC07_1LDC1L - Power Supply 24VDC - Spare

       CALL #"PLC1.1_DC07_1LDC1L"
       (
         CM_No := 458 ,
         Tab := 13 ,
         SubTab := 1 ,
         CfgType := 0 ,
         CfgInvert := True ,
         InputRaw := PLC1_DC07_1LDC1L_DI_Flt ,
         SC_Local := SL_13 ,
         CM_ALM := #ALM[449] ,
       );

NETWORK
TITLE = 459 - PLC1.1_DC07_2LDC2L - Power Supply 24VDC - Spare

       CALL #"PLC1.1_DC07_2LDC2L"
       (
         CM_No := 459 ,
         Tab := 13 ,
         SubTab := 1 ,
         CfgType := 0 ,
         CfgInvert := True ,
         InputRaw := PLC1_DC07_2LDC2L_DI_Flt ,
         SC_Local := SL_13 ,
         CM_ALM := #ALM[450] ,
       );

NETWORK
TITLE = 460 - PLC1.1_DC07_3LDC3L - Power Supply 24VDC - Spare

       CALL #"PLC1.1_DC07_3LDC3L"
       (
         CM_No := 460 ,
         Tab := 13 ,
         SubTab := 1 ,
         CfgType := 0 ,
         CfgInvert := True ,
         InputRaw := PLC1_DC07_3LDC3L_DI_Flt ,
         SC_Local := SL_13 ,
         CM_ALM := #ALM[451] ,
       );

NETWORK
TITLE = 461 - PLC1.1_DC07_4LDC4L - Power Supply 24VDC - Spare

       CALL #"PLC1.1_DC07_4LDC4L"
       (
         CM_No := 461 ,
         Tab := 13 ,
         SubTab := 1 ,
         CfgType := 0 ,
         CfgInvert := True ,
         InputRaw := PLC1_DC07_4LDC4L_DI_Flt ,
         SC_Local := SL_13 ,
         CM_ALM := #ALM[452] ,
       );

NETWORK
TITLE = 462 - PLC1.1_PLC1_KF1001 - L83ES PLC1 - Master - VLAN 2221 - Slot 0

       CALL #"PLC1.1_PLC1_KF1001"
       (
         CM_No := 462 ,
         Tab := 13 ,
         SubTab := 1 ,
         CfgType := 0 ,
         CfgInvert := True ,
         InputRaw :=  ,
         SC_Local := SL_13 ,
         CM_ALM := #ALM[453] ,
       );

NETWORK
TITLE = 463 - PLC1.1_PLC1_KF1002 - EN4TR - VLAN 2220 - Slot 1

       CALL #"PLC1.1_PLC1_KF1002"
       (
         CM_No := 463 ,
         Tab := 13 ,
         SubTab := 1 ,
         CfgType := 0 ,
         CfgInvert := True ,
         InputRaw :=  ,
         SC_Local := SL_13 ,
         CM_ALM := #ALM[454] ,
       );

NETWORK
TITLE = 464 - PLC1.1_PLC1_KF1003 - L81ES PLC2  - VLAN 2222 - Slot 2

       CALL #"PLC1.1_PLC1_KF1003"
       (
         CM_No := 464 ,
         Tab := 13 ,
         SubTab := 1 ,
         CfgType := 0 ,
         CfgInvert := True ,
         InputRaw :=  ,
         SC_Local := SL_13 ,
         CM_ALM := #ALM[455] ,
       );

NETWORK
TITLE = 465 - PLC1.1_PLC1_KF1005 - EN2T - VLAN 2224 - Slot 4

       CALL #"PLC1.1_PLC1_KF1005"
       (
         CM_No := 465 ,
         Tab := 13 ,
         SubTab := 1 ,
         CfgType := 0 ,
         CfgInvert := True ,
         InputRaw :=  ,
         SC_Local := SL_13 ,
         CM_ALM := #ALM[456] ,
       );

NETWORK
TITLE = 466 - PLC1.1_Din_SP01 - Spare Digital Input - nan

       CALL #"PLC1.1_Din_SP01"
       (
         CM_No := 466 ,
         Tab := 13 ,
         SubTab := 1 ,
         CfgType := 0 ,
         CfgInvert := True ,
         InputRaw := PLC1_Din_SP01_DI_Disp ,
         SC_Local := SL_13 ,
         CM_ALM := #ALM[457] ,
       );

NETWORK
TITLE = 467 - PLC1.1_IO_KF1000 - Point IO - EtherNet/IP Adapter

       CALL #"PLC1.1_IO_KF1000"
       (
         CM_No := 467 ,
         Tab := 13 ,
         SubTab := 1 ,
         CfgType := 0 ,
         CfgInvert := True ,
         InputRaw :=  ,
         SC_Local := SL_13 ,
         CM_ALM := #ALM[458] ,
       );

NETWORK
TITLE = 468 - PLC2.1_AC01_FC2010 - 115VAC Power Supply - Circuit Breaker

       CALL #"PLC2.1_AC01_FC2010"
       (
         CM_No := 468 ,
         Tab := 13 ,
         SubTab := 2 ,
         CfgType := 0 ,
         CfgInvert := True ,
         InputRaw := PLC2_AC01_FC2010_DI_Flt ,
         SC_Local := SL_13 ,
         CM_ALM := #ALM[459] ,
       );

NETWORK
TITLE = 469 - PLC2.1_AC02_FC2010 - 24VAC Power Supply - Circuit Breaker

       CALL #"PLC2.1_AC02_FC2010"
       (
         CM_No := 469 ,
         Tab := 13 ,
         SubTab := 2 ,
         CfgType := 0 ,
         CfgInvert := True ,
         InputRaw := PLC2_AC02_FC2010_DI_Flt ,
         SC_Local := SL_13 ,
         CM_ALM := #ALM[460] ,
       );

NETWORK
TITLE = 470 - PLC2.1_A711_FC1790 - Power Supply 24VAC - Nozzle Supply

       CALL #"PLC2.1_A711_FC1790"
       (
         CM_No := 470 ,
         Tab := 13 ,
         SubTab := 2 ,
         CfgType := 0 ,
         CfgInvert := True ,
         InputRaw := PLC2_A711_FC1790_DI_Flt ,
         SC_Local := SL_13 ,
         CM_ALM := #ALM[461] ,
       );

NETWORK
TITLE = 471 - PLC2.1_A712_FC1791 - Power Supply 24VAC - Nozzle Supply

       CALL #"PLC2.1_A712_FC1791"
       (
         CM_No := 471 ,
         Tab := 13 ,
         SubTab := 2 ,
         CfgType := 0 ,
         CfgInvert := True ,
         InputRaw := PLC2_A712_FC1791_DI_Flt ,
         SC_Local := SL_13 ,
         CM_ALM := #ALM[462] ,
       );

NETWORK
TITLE = 472 - PLC2.1_AC02_FC2011 - 24VAC Power Supply - Circuit Breaker

       CALL #"PLC2.1_AC02_FC2011"
       (
         CM_No := 472 ,
         Tab := 13 ,
         SubTab := 2 ,
         CfgType := 0 ,
         CfgInvert := True ,
         InputRaw := PLC2_AC02_FC2011_DI_Flt ,
         SC_Local := SL_13 ,
         CM_ALM := #ALM[463] ,
       );

NETWORK
TITLE = 473 - PLC2.1_A721_FC1792 - Power Supply 24VAC - Nozzle Supply

       CALL #"PLC2.1_A721_FC1792"
       (
         CM_No := 473 ,
         Tab := 13 ,
         SubTab := 2 ,
         CfgType := 0 ,
         CfgInvert := True ,
         InputRaw := PLC2_A721_FC1792_DI_Flt ,
         SC_Local := SL_13 ,
         CM_ALM := #ALM[464] ,
       );

NETWORK
TITLE = 474 - PLC2.1_A722_FC1793 - Power Supply 24VAC - Nozzle Supply

       CALL #"PLC2.1_A722_FC1793"
       (
         CM_No := 474 ,
         Tab := 13 ,
         SubTab := 2 ,
         CfgType := 0 ,
         CfgInvert := True ,
         InputRaw := PLC2_A722_FC1793_DI_Flt ,
         SC_Local := SL_13 ,
         CM_ALM := #ALM[465] ,
       );

NETWORK
TITLE = 475 - PLC2.1_AC02_FC2012 - 24VAC Power Supply - Circuit Breaker

       CALL #"PLC2.1_AC02_FC2012"
       (
         CM_No := 475 ,
         Tab := 13 ,
         SubTab := 2 ,
         CfgType := 0 ,
         CfgInvert := True ,
         InputRaw := PLC2_AC02_FC2012_DI_Flt ,
         SC_Local := SL_13 ,
         CM_ALM := #ALM[466] ,
       );

NETWORK
TITLE = 476 - PLC2.1_A731_FC1794 - Power Supply 24VAC - Nozzle Supply

       CALL #"PLC2.1_A731_FC1794"
       (
         CM_No := 476 ,
         Tab := 13 ,
         SubTab := 2 ,
         CfgType := 0 ,
         CfgInvert := True ,
         InputRaw := PLC2_A731_FC1794_DI_Flt ,
         SC_Local := SL_13 ,
         CM_ALM := #ALM[467] ,
       );

NETWORK
TITLE = 477 - PLC2.1_A732_FC1795 - Power Supply 24VAC - Nozzle Supply

       CALL #"PLC2.1_A732_FC1795"
       (
         CM_No := 477 ,
         Tab := 13 ,
         SubTab := 2 ,
         CfgType := 0 ,
         CfgInvert := True ,
         InputRaw := PLC2_A732_FC1795_DI_Flt ,
         SC_Local := SL_13 ,
         CM_ALM := #ALM[468] ,
       );

NETWORK
TITLE = 478 - PLC2.1_DC01_FC1010 - Power Feed Module 24VDC - Status

       CALL #"PLC2.1_DC01_FC1010"
       (
         CM_No := 478 ,
         Tab := 13 ,
         SubTab := 2 ,
         CfgType := 0 ,
         CfgInvert := True ,
         InputRaw := PLC2_DC01_FC1010_DI_Sts ,
         SC_Local := SL_13 ,
         CM_ALM := #ALM[469] ,
       );

NETWORK
TITLE = 479 - PLC2.1_DC02_1LDC1L - Power Supply 24VDC - MCC2

       CALL #"PLC2.1_DC02_1LDC1L"
       (
         CM_No := 479 ,
         Tab := 13 ,
         SubTab := 2 ,
         CfgType := 0 ,
         CfgInvert := True ,
         InputRaw := PLC2_DC02_1LDC1L_DI_Flt ,
         SC_Local := SL_13 ,
         CM_ALM := #ALM[470] ,
       );

NETWORK
TITLE = 480 - PLC2.1_DC02_2LDC2L - Power Supply 24VDC - LCP20 / OP20

       CALL #"PLC2.1_DC02_2LDC2L"
       (
         CM_No := 480 ,
         Tab := 13 ,
         SubTab := 2 ,
         CfgType := 0 ,
         CfgInvert := True ,
         InputRaw := PLC2_DC02_2LDC2L_DI_Flt ,
         SC_Local := SL_13 ,
         CM_ALM := #ALM[471] ,
       );

NETWORK
TITLE = 481 - PLC2.1_DC02_3LDC3L - Power Supply 24VDC - Spare

       CALL #"PLC2.1_DC02_3LDC3L"
       (
         CM_No := 481 ,
         Tab := 13 ,
         SubTab := 2 ,
         CfgType := 0 ,
         CfgInvert := True ,
         InputRaw := PLC2_DC02_3LDC3L_DI_Flt ,
         SC_Local := SL_13 ,
         CM_ALM := #ALM[472] ,
       );

NETWORK
TITLE = 482 - PLC2.1_DC03_1LDC1L - Power Supply 24VDC - MCC3

       CALL #"PLC2.1_DC03_1LDC1L"
       (
         CM_No := 482 ,
         Tab := 13 ,
         SubTab := 2 ,
         CfgType := 0 ,
         CfgInvert := True ,
         InputRaw := PLC2_DC03_1LDC1L_DI_Flt ,
         SC_Local := SL_13 ,
         CM_ALM := #ALM[473] ,
       );

NETWORK
TITLE = 483 - PLC2.1_DC03_2LDC2L - Power Supply 24VDC - LCP30 / OP30

       CALL #"PLC2.1_DC03_2LDC2L"
       (
         CM_No := 483 ,
         Tab := 13 ,
         SubTab := 2 ,
         CfgType := 0 ,
         CfgInvert := True ,
         InputRaw := PLC2_DC03_2LDC2L_DI_Flt ,
         SC_Local := SL_13 ,
         CM_ALM := #ALM[474] ,
       );

NETWORK
TITLE = 484 - PLC2.1_DC03_3LDC3L - Power Supply 24VDC - Spare

       CALL #"PLC2.1_DC03_3LDC3L"
       (
         CM_No := 484 ,
         Tab := 13 ,
         SubTab := 2 ,
         CfgType := 0 ,
         CfgInvert := True ,
         InputRaw := PLC2_DC03_3LDC3L_DI_Flt ,
         SC_Local := SL_13 ,
         CM_ALM := #ALM[475] ,
       );

NETWORK
TITLE = 485 - PLC2.1_DC04_1LDC1L - Power Supply 24VDC - MCC4

       CALL #"PLC2.1_DC04_1LDC1L"
       (
         CM_No := 485 ,
         Tab := 13 ,
         SubTab := 2 ,
         CfgType := 0 ,
         CfgInvert := True ,
         InputRaw := PLC2_DC04_1LDC1L_DI_Flt ,
         SC_Local := SL_13 ,
         CM_ALM := #ALM[476] ,
       );

NETWORK
TITLE = 486 - PLC2.1_DC04_2LDC2L - Power Supply 24VDC - LCP40 / OP40

       CALL #"PLC2.1_DC04_2LDC2L"
       (
         CM_No := 486 ,
         Tab := 13 ,
         SubTab := 2 ,
         CfgType := 0 ,
         CfgInvert := True ,
         InputRaw := PLC2_DC04_2LDC2L_DI_Flt ,
         SC_Local := SL_13 ,
         CM_ALM := #ALM[477] ,
       );

NETWORK
TITLE = 487 - PLC2.1_DC04_3LDC3L - Power Supply 24VDC - Spare

       CALL #"PLC2.1_DC04_3LDC3L"
       (
         CM_No := 487 ,
         Tab := 13 ,
         SubTab := 2 ,
         CfgType := 0 ,
         CfgInvert := True ,
         InputRaw := PLC2_DC04_3LDC3L_DI_Flt ,
         SC_Local := SL_13 ,
         CM_ALM := #ALM[478] ,
       );

NETWORK
TITLE = 488 - PLC2.1_DC05_1LDC1L - Power Supply 24VDC - MCC5

       CALL #"PLC2.1_DC05_1LDC1L"
       (
         CM_No := 488 ,
         Tab := 13 ,
         SubTab := 2 ,
         CfgType := 0 ,
         CfgInvert := True ,
         InputRaw := PLC2_DC05_1LDC1L_DI_Flt ,
         SC_Local := SL_13 ,
         CM_ALM := #ALM[479] ,
       );

NETWORK
TITLE = 489 - PLC2.1_DC05_2LDC2L - Power Supply 24VDC - Spare

       CALL #"PLC2.1_DC05_2LDC2L"
       (
         CM_No := 489 ,
         Tab := 13 ,
         SubTab := 2 ,
         CfgType := 0 ,
         CfgInvert := True ,
         InputRaw := PLC2_DC05_2LDC2L_DI_Flt ,
         SC_Local := SL_13 ,
         CM_ALM := #ALM[480] ,
       );

NETWORK
TITLE = 490 - PLC2.1_DC05_3LDC3L - Power Supply 24VDC - LCP52 / OP52 / PNEU52

       CALL #"PLC2.1_DC05_3LDC3L"
       (
         CM_No := 490 ,
         Tab := 13 ,
         SubTab := 2 ,
         CfgType := 0 ,
         CfgInvert := True ,
         InputRaw := PLC2_DC05_3LDC3L_DI_Flt ,
         SC_Local := SL_13 ,
         CM_ALM := #ALM[481] ,
       );

NETWORK
TITLE = 491 - PLC2.1_DC06_1LDC1L - Power Supply 24VDC - MCC6

       CALL #"PLC2.1_DC06_1LDC1L"
       (
         CM_No := 491 ,
         Tab := 13 ,
         SubTab := 2 ,
         CfgType := 0 ,
         CfgInvert := True ,
         InputRaw := PLC2_DC06_1LDC1L_DI_Flt ,
         SC_Local := SL_13 ,
         CM_ALM := #ALM[482] ,
       );

NETWORK
TITLE = 492 - PLC2.1_DC06_2LDC2L - Power Supply 24VDC - LCP61 / OP61 / PNEU61

       CALL #"PLC2.1_DC06_2LDC2L"
       (
         CM_No := 492 ,
         Tab := 13 ,
         SubTab := 2 ,
         CfgType := 0 ,
         CfgInvert := True ,
         InputRaw := PLC2_DC06_2LDC2L_DI_Flt ,
         SC_Local := SL_13 ,
         CM_ALM := #ALM[483] ,
       );

NETWORK
TITLE = 493 - PLC2.1_DC06_3LDC3L - Power Supply 24VDC - LCP62 / OP62 / PNEU62

       CALL #"PLC2.1_DC06_3LDC3L"
       (
         CM_No := 493 ,
         Tab := 13 ,
         SubTab := 2 ,
         CfgType := 0 ,
         CfgInvert := True ,
         InputRaw := PLC2_DC06_3LDC3L_DI_Flt ,
         SC_Local := SL_13 ,
         CM_ALM := #ALM[484] ,
       );

NETWORK
TITLE = 494 - PLC2.1_DC07_1LDC1L - Power Supply 24VDC - MCC7

       CALL #"PLC2.1_DC07_1LDC1L"
       (
         CM_No := 494 ,
         Tab := 13 ,
         SubTab := 2 ,
         CfgType := 0 ,
         CfgInvert := True ,
         InputRaw := PLC2_DC07_1LDC1L_DI_Flt ,
         SC_Local := SL_13 ,
         CM_ALM := #ALM[485] ,
       );

NETWORK
TITLE = 495 - PLC2.1_DC07_2LDC2L - Power Supply 24VDC - LCP71

       CALL #"PLC2.1_DC07_2LDC2L"
       (
         CM_No := 495 ,
         Tab := 13 ,
         SubTab := 2 ,
         CfgType := 0 ,
         CfgInvert := True ,
         InputRaw := PLC2_DC07_2LDC2L_DI_Flt ,
         SC_Local := SL_13 ,
         CM_ALM := #ALM[486] ,
       );

NETWORK
TITLE = 496 - PLC2.1_DC07_3LDC3L - Power Supply 24VDC - LCP72 / OP72

       CALL #"PLC2.1_DC07_3LDC3L"
       (
         CM_No := 496 ,
         Tab := 13 ,
         SubTab := 2 ,
         CfgType := 0 ,
         CfgInvert := True ,
         InputRaw := PLC2_DC07_3LDC3L_DI_Flt ,
         SC_Local := SL_13 ,
         CM_ALM := #ALM[487] ,
       );

NETWORK
TITLE = 497 - PLC2.1_DC08_1LDC1L - Power Supply 24VDC - MCC8

